_EvaluateCompletionConditions();

_CommandsCyclic();

IF FirstCycScan THEN
	_ComponentCyclic();
	FirstCycScan	:= FALSE;
END_IF

_UpdateBusyStatus();

_UpdateComponentStatus();

HMICommunication(); //Keeps the HMI data up to date, and processes requests from the HMI for this component
END_METHOD

END_FUNCTION_BLOCK

// Configuration/FB_CmdPermIntlkConfiguration
{attribute 'no_explicit_call' := 'do not call this POU directly'}
FUNCTION_BLOCK FB_CmdPermIntlkConfiguration EXTENDS FB_BaseStatic IMPLEMENTS I_CommandConfiguration, I_PermIntlkConfiguration
VAR
	PermIntlkConfiguration		: ST_PermIntlkConfiguration;
	CommandConfiguration		: ST_CommandConfiguration;
END_VAR

METHOD PROTECTED _InitializeReferences : BOOL
//Order is important!
BaseConfiguration.InstancePath 				REF= SUPER^.InstancePath;

PermIntlkConfiguration.BaseConfiguration 	REF= SUPER^.BaseConfiguration;
CommandConfiguration.BaseConfiguration		REF= SUPER^.BaseConfiguration;

CommandConfiguration.PermIntlkConfiguration REF= PermIntlkConfiguration;
                                	
_InitializeReferences 						:= TRUE; // apply at end of all reference initialization
END_METHOD

PROPERTY P_CommandConfiguration : REFERENCE TO ST_CommandConfiguration
GET
P_CommandConfiguration REF= CommandConfiguration;
END_GET
END_PROPERTY

PROPERTY P_PermIntlkConfiguration : REFERENCE TO ST_PermIntlkConfiguration
GET
P_PermIntlkConfiguration REF= PermIntlkConfiguration;
END_GET
END_PROPERTY

END_FUNCTION_BLOCK

// RingBuffer/POUs/FB_RingBufferICmd
{attribute 'no_explicit_call' := 'do not call this POU directly'}
FUNCTION_BLOCK FB_RingBufferICmd EXTENDS FB_RingBufferBase IMPLEMENTS I_RingBufferBase, I_RingBufferICmd
VAR
  Buffer              	: ARRAY[GPL_RingBuffer.MIN_NUMBER_OBJECTS..GPL_RingBuffer.MAX_NUMBER_OBJECTS] OF ST_SystimeICmd;
  LastObjRemoved		: ST_SystimeICmd;
  LastObjPeeked			: ST_SystimeICmd;
  LastObjRead			: ST_SystimeICmd;
END_VAR

METHOD ClearLastRemoved
MEMSET(destAddr := ADR(LastObjRemoved), fillByte := 16#00, n := RingBufferConfiguration.ByteCountOfDataObj);
END_METHOD

PROPERTY P_RingBufferStatus : REFERENCE TO ST_RingBufferStatus
GET
P_RingBufferStatus REF= SUPER^.RingBufferStatus;
END_GET
END_PROPERTY

METHOD PUBLIC RemoveObject
VAR_OUTPUT
    Error : BOOL;
END_VAR
VAR
    ByteSize : UDINT;
    Addr     : PVOID;
END_VAR
Error := FALSE;
ByteSize := RingBufferConfiguration.ByteCountOfDataObj;

IF RingBufferStatus.ObjectCountInBufferPrim = 0 THEN   (* nothing to pop *)
    Error := TRUE;
    RETURN;
END_IF;

Addr := pBufferStart +
        (RemoveIncrement MOD RingBufferStatus.BufferCapacity) * ByteSize;

IF Tc2_System.MEMMOVE(srcAddr := Addr, destAddr := ADR(LastObjRemoved), n := ByteSize) <> ByteSize THEN
    Error := TRUE;
    RETURN;
END_IF;
Tc2_System.MEMSET(destAddr := Addr, fillByte := 16#00, n := ByteSize);

(* advance remove side *)
RemoveIncrement := RemoveIncrement + 1;
RemoveIndex     := (RemoveIncrement MOD RingBufferStatus.BufferCapacity)
                 + GPL_RingBuffer.MIN_NUMBER_OBJECTS;
pRemove         := pBufferStart +
                   (RemoveIncrement MOD RingBufferStatus.BufferCapacity) * ByteSize;

(* counters / flags *)
RingBufferStatus.ObjectCountInBufferPrim := RingBufferStatus.ObjectCountInBufferPrim - 1;
IF RingBufferStatus.GlobalCounter > 0 THEN
    RingBufferStatus.GlobalCounter := RingBufferStatus.GlobalCounter - 1;
END_IF;

RingBufferStatus.ObjectWasRemovedPrimary := TRUE;

RingBufferStatus.Overwriting  := FALSE;                                 (* we freed space *)
RingBufferStatus.WillOverwrite :=                                     (* preview for next cycle *)
    (RingBufferStatus.ObjectCountInBufferPrim = RingBufferStatus.BufferCapacity);

(* derived *)
RingBufferStatus.BufferIsFullPrim :=
    (RingBufferStatus.ObjectCountInBufferPrim = RingBufferStatus.BufferCapacity);
RingBufferStatus.ByteCountInBufferPrim :=
    RingBufferStatus.ObjectCountInBufferPrim * ByteSize;
END_METHOD

METHOD PUBLIC AddObject
VAR_INPUT
    RefObject : REFERENCE TO ST_SystimeICmd;
END_VAR
VAR_OUTPUT
    Error : BOOL;
END_VAR
VAR
    ByteSize   : UDINT;
    ByteOffset : UDINT;
    WriteAddr  : PVOID;
END_VAR
Error := FALSE;
ByteSize := RingBufferConfiguration.ByteCountOfDataObj;

(* ---------- GUARDS ---------- *)
IF (RingBufferStatus.BufferCapacity = 0) OR (NOT __ISVALIDREF(RefObject)) THEN
    Error := TRUE;                           (* zero-capacity or bogus ref *)
    RETURN;
END_IF;

(* ---------- PREDICT / PREP ---------- *)
RingBufferStatus.WillOverwrite :=
    (RingBufferStatus.ObjectCountInBufferPrim >= RingBufferStatus.BufferCapacity);

ByteOffset := (WriteIncrement MOD RingBufferStatus.BufferCapacity) * ByteSize;
WriteAddr  := pBufferStart + ByteOffset;

(* ---------- WRITE ---------- *)
RefObject.systimestamp := Tc2_System.F_GetSystemTime();
IF Tc2_System.MEMMOVE(srcAddr := ADR(RefObject), destAddr := WriteAddr, n := ByteSize) <> ByteSize THEN
    Error := TRUE;
    RETURN;
END_IF;

(* ---------- ADVANCE WRITE POINTERS ---------- *)
WriteIncrement := WriteIncrement + 1;
WriteIndex := (WriteIncrement MOD RingBufferStatus.BufferCapacity)
            + GPL_RingBuffer.MIN_NUMBER_OBJECTS;

(* ---------- COUNTERS & FLAGS ---------- *)
IF RingBufferStatus.WillOverwrite THEN
    (* buffer is full – push remove side forward one slot *)
    RemoveIncrement := RemoveIncrement + 1;
    pRemove := pBufferStart
             + (RemoveIncrement MOD RingBufferStatus.BufferCapacity) * ByteSize;
    RingBufferStatus.Overwriting := TRUE;              (* occurred *this* cycle *)
ELSE
    RingBufferStatus.ObjectCountInBufferPrim := RingBufferStatus.ObjectCountInBufferPrim + 1;
    RingBufferStatus.GlobalCounter           := RingBufferStatus.GlobalCounter + 1;
    RingBufferStatus.Overwriting             := FALSE;
END_IF;

RingBufferStatus.ObjectWasAddedPrimary := TRUE;

(* ---------- STATE FOR NEXT SCAN ---------- *)
RingBufferStatus.WillOverwrite :=
    (RingBufferStatus.ObjectCountInBufferPrim >= RingBufferStatus.BufferCapacity);

(* ---------- DERIVED VALUES ---------- *)
RingBufferStatus.BufferIsFullPrim :=
    (RingBufferStatus.ObjectCountInBufferPrim = RingBufferStatus.BufferCapacity);
RingBufferStatus.ByteCountInBufferPrim :=
    RingBufferStatus.ObjectCountInBufferPrim * ByteSize;
END_METHOD

PROPERTY P_Buffer : REFERENCE TO ARRAY[GPL_RingBuffer.MIN_NUMBER_OBJECTS..GPL_RingBuffer.MAX_NUMBER_OBJECTS] OF ST_SystimeICmd;
GET
P_Buffer REF= Buffer;
END_GET
END_PROPERTY

PROPERTY P_LastObjectPeeked : REFERENCE TO ST_SystimeICmd
GET
P_LastObjectPeeked REF= LastObjPeeked;
END_GET
END_PROPERTY

PROPERTY P_LastObjectRead : REFERENCE TO ST_SystimeICmd
GET
P_LastObjectRead REF= LastObjRead;
END_GET
END_PROPERTY

PROPERTY P_LastObjectRemoved : REFERENCE TO ST_SystimeICmd
GET
P_LastObjectRemoved REF= LastObjRemoved;
END_GET
END_PROPERTY

METHOD PUBLIC PeekObject : ST_SystimeICmd
PeekIndex := (RemoveIncrement MOD SUPER^.RingBufferStatus.BufferCapacity) + GPL_RingBuffer.MIN_NUMBER_OBJECTS;
PeekAddr := pBufferStart + (PeekIndex - GPL_RingBuffer.MIN_NUMBER_OBJECTS) * RingBufferConfiguration.ByteCountOfDataObj;

// Step 2: Conditional peek (non-mutating)
IF SUPER^.RingBufferStatus.GlobalCounter > 0 THEN
    SUPER^.RingBufferStatus.CountBytesPeeked := Tc2_System.MEMMOVE(
        srcAddr := PeekAddr,
        destAddr := ADR(LastObjPeeked),
        n := RingBufferConfiguration.ByteCountOfDataObj
    );

    IF SUPER^.RingBufferStatus.CountBytesPeeked > 0 THEN
        RingBufferStatus.ObjectWasPeekedPrimary := TRUE;
		PeekObject	:= LastObjPeeked;
    END_IF
ELSE
    RingBufferStatus.ObjectWasPeekedPrimary := FALSE;
    //LastObjPeeked.stringval := '';
END_IF
END_METHOD

METHOD ReadObject : ST_SystimeICmd
VAR_OUTPUT
  Error : BOOL;
END_VAR
// Step 1: Check if buffer has data
IF SUPER^.RingBufferStatus.GlobalCounter > 0 THEN

    // Step 2: Calculate read offset and pointer
    RingBufferConfiguration.ReadByteOffset := (RemoveIncrement MOD RingBufferStatus.BufferCapacity) * RingBufferConfiguration.ByteCountOfDataObj;
    ReadAddr := pBufferStart + RingBufferConfiguration.ReadByteOffset;

    // Step 3: Read memory
    SUPER^.RingBufferStatus.CountBytesRead := Tc2_System.MEMMOVE(
        srcAddr := ReadAddr,
        destAddr := ADR(LastObjRead),
        n := RingBufferConfiguration.ByteCountOfDataObj
    );

    // Step 4: Handle result
    IF SUPER^.RingBufferStatus.CountBytesRead = RingBufferConfiguration.ByteCountOfDataObj THEN
        RingBufferStatus.ObjectWasReadPrimary := TRUE;

        RemoveIncrement := RemoveIncrement + 1;

        // Update index and pRemove based on RemoveIncrement
        RemoveIndex := (RemoveIncrement MOD RingBufferStatus.BufferCapacity)
                       + GPL_RingBuffer.MIN_NUMBER_OBJECTS;

        pRemove := pBufferStart + 
                   (RemoveIncrement MOD RingBufferStatus.BufferCapacity) * RingBufferConfiguration.ByteCountOfDataObj;

        SUPER^.RingBufferStatus.GlobalCounter := SUPER^.RingBufferStatus.GlobalCounter - 1;
    ELSE
        RingBufferStatus.ObjectWasReadPrimary := FALSE;
        //LastObjRead.stringval := ''; // 🛠 Corrected
        Error := TRUE;
    END_IF
ELSE
    RingBufferStatus.ObjectWasReadPrimary := FALSE;
    //LastObjRead.stringval := ''; // 🛠 Corrected
    Error := TRUE;
END_IF

UpdateObjectCtInBuffers();
END_METHOD

METHOD PROTECTED UpdateRemovePointer
VAR_INPUT
  pRemovePtr  : PVOID;
END_VAR
pRemove := ADR(Buffer[RemoveIndex]);

pRemoveUpdated  := TRUE;
END_METHOD

METHOD PROTECTED UpdateWritePointer
VAR_INPUT
  pWritePtr  : PVOID;
END_VAR
IF (WriteIndex = GPL_RingBuffer.MIN_NUMBER_OBJECTS) THEN
  pWrite        := ADR(Buffer[GPL_RingBuffer.MIN_NUMBER_OBJECTS]);
ELSIF (WriteIndex > GPL_RingBuffer.MIN_NUMBER_OBJECTS) AND 
  (WriteIndex <= GPL_RingBuffer.MAX_NUMBER_OBJECTS) THEN
  pWrite        := IncrementPointer(pPointer  := pWrite, ByteCtIncrement := RingBufferConfiguration.ByteCountOfDataObj);
END_IF

pWriteUpdated   := TRUE;
END_METHOD

(* Basic component initialization logic*)
METHOD PROTECTED _Initialize : BOOL
VAR
	InterimInit : BOOL;
END_VAR
InterimInit := _InitializeChildrenDependencies();

InterimInit	:= _InitializeReferences();

IF NOT InterimInit THEN
	IF SUPER^.BaseConfiguration.LogTraceConfiguration.What.xLogToEventLogger THEN
		TraceWithSeverity(Message := Tc2_Standard.CONCAT('Initialization Failed at ', __POUNAME()), Severity := Global.TcEventSeverity.Error);
	END_IF
END_IF

RingBufferStatus.BufferCapacity  := (GPL_RingBuffer.MAX_NUMBER_OBJECTS - GPL_RingBuffer.MIN_NUMBER_OBJECTS) +1;

RemoveIndex  := GPL_RingBuffer.MIN_NUMBER_OBJECTS;
PeekIndex	 := GPL_RingBuffer.MIN_NUMBER_OBJECTS;

pBufferStart	:= ADR(Buffer[GPL_RingBuffer.MIN_NUMBER_OBJECTS]);

RingBufferConfiguration.ByteCountOfDataObj      := SIZEOF(Buffer[GPL_RingBuffer.MIN_NUMBER_OBJECTS]);

IF (pWrite = Tc3_Module.NULL) THEN
  pWrite  := ADR(Buffer[GPL_RingBuffer.MIN_NUMBER_OBJECTS]);
END_IF

IF (pRemove = Tc3_Module.NULL) THEN
  pRemove  := ADR(Buffer[GPL_RingBuffer.MIN_NUMBER_OBJECTS]);
END_IF

InterimInit	:= _SetDependencyConfiguration();

_Initialize 	:= InterimInit;
END_METHOD

METHOD ClearBuffer
MEMSET(destAddr := ADR(Buffer[GPL_RingBuffer.MIN_NUMBER_OBJECTS]), fillByte := 16#00, n := (RingBufferConfiguration.ByteCountOfDataObj*SUPER^.RingBufferStatus.BufferCapacity));

WriteIncrement := 0;
RemoveIncrement := 0;
SUPER^.RingBufferStatus.GlobalCounter := 0;
pWrite := ADR(Buffer[GPL_RingBuffer.MIN_NUMBER_OBJECTS]);
pRemove := ADR(Buffer[GPL_RingBuffer.MIN_NUMBER_OBJECTS]);
UpdateObjectCtInBuffers();
END_METHOD

END_FUNCTION_BLOCK

// RingBuffer/POUs/FB_RingBufferBase
FUNCTION_BLOCK ABSTRACT FB_RingBufferBase EXTENDS FB_BaseStatic
VAR
	RingBufferConfiguration    		: ST_RingBufferCfg;
	pRemove        					: PVOID;
	pWrite         					: PVOID;
	pBufferStart					: PVOID;
	RemoveAddr 						: PVOID;
	PeekAddr						: PVOID;
	ReadAddr						: PVOID;
	pRemoveUpdated 					: BOOL;
	pWriteUpdated  					: BOOL;
	WriteIncrement 					: UDINT;
	RemoveIncrement					: UDINT;
	WriteIndex     					: UDINT;
	RemoveIndex    					: UDINT;
	PeekIndex						: UDINT;
	ReadIndex						: UDINT;
	RingBufferStatus				: ST_RingBufferStatus;
END_VAR

(* Basic component initialization logic*)
METHOD PROTECTED _Initialize : BOOL
VAR
	InterimInit : BOOL;
END_VAR
// Initialize children dependencies first
InterimInit := _InitializeChildrenDependencies();
IF NOT InterimInit THEN
	IF BaseConfiguration.LogTraceConfiguration.What.xLogToEventLogger AND NOT BaseStatus.LogTraceStatus.InitChildrenFailureShown THEN
		TraceWithSeverity(Message := Tc2_Standard.CONCAT('_InitializeChildrenDependencies Failed at ', __POUNAME()), Severity := Global.TcEventSeverity.Error);
		BaseStatus.LogTraceStatus.InitChildrenFailureShown := TRUE;
	END_IF
	_Initialize := FALSE;
	RETURN;
END_IF

// Initialize references second
InterimInit := _InitializeReferences();
IF NOT InterimInit THEN
	IF BaseConfiguration.LogTraceConfiguration.What.xLogToEventLogger AND NOT BaseStatus.LogTraceStatus.InitReferencesFailureShown THEN
		TraceWithSeverity(Message := Tc2_Standard.CONCAT('_InitializeReferences Failed at ', __POUNAME()), Severity := Global.TcEventSeverity.Error);
		BaseStatus.LogTraceStatus.InitReferencesFailureShown := TRUE;
	END_IF
	_Initialize := FALSE;
	RETURN;
END_IF

// Set buffer-specific initialization values
RingBufferStatus.BufferCapacity := (GPL_RingBuffer.MAX_NUMBER_OBJECTS - GPL_RingBuffer.MIN_NUMBER_OBJECTS) + 1;
RemoveIndex := GPL_RingBuffer.MIN_NUMBER_OBJECTS;
PeekIndex := GPL_RingBuffer.MIN_NUMBER_OBJECTS;

// Set dependency configuration last
InterimInit := _SetDependencyConfiguration();
IF NOT InterimInit THEN
	IF BaseConfiguration.LogTraceConfiguration.What.xLogToEventLogger AND NOT BaseStatus.LogTraceStatus.InitDependencyConfigFailureShown THEN
		TraceWithSeverity(Message := Tc2_Standard.CONCAT('_SetDependencyConfiguration Failed at ', __POUNAME()), Severity := Global.TcEventSeverity.Error);
		BaseStatus.LogTraceStatus.InitDependencyConfigFailureShown := TRUE;
	END_IF
	_Initialize := FALSE;
	RETURN;
END_IF

// All initialization steps succeeded
_Initialize := TRUE;
END_METHOD

METHOD PROTECTED _InitializeReferences : BOOL
//Order is important!
BaseConfiguration.InstancePath 				REF= SUPER^.InstancePath;

RingBufferConfiguration.BaseConfiguration	REF= SUPER^.BaseConfiguration;

RingBufferStatus.BaseStatus					REF= SUPER^.BaseStatus;

_InitializeReferences 						:= TRUE;
END_METHOD

METHOD PROTECTED UpdateObjectCtInBuffers
RingBufferStatus.BufferIsFullPrim :=
    (RingBufferStatus.ObjectCountInBufferPrim = RingBufferStatus.BufferCapacity);
RingBufferStatus.ByteCountInBufferPrim :=
    RingBufferStatus.ObjectCountInBufferPrim * RingBufferConfiguration.ByteCountOfDataObj;
END_METHOD

PROPERTY P_ObjCountInBuffer : ULINT
GET
P_ObjCountInBuffer  := RingBufferStatus.ObjectCountInBufferPrim;
END_GET
END_PROPERTY

PROPERTY P_ObjectWasAdded : REFERENCE TO BOOL
GET
//P_ObjectWasAdded REF= RingBufferStatus.ObjectWasAddedPrimary;
P_ObjectWasAdded REF= RingBufferStatus.ObjectWasAddedPrimary;
END_GET
END_PROPERTY

PROPERTY P_ObjectWasPeeked : REFERENCE TO BOOL
GET
P_ObjectWasPeeked REF= RingBufferStatus.ObjectWasPeekedPrimary;
END_GET
END_PROPERTY

PROPERTY P_ObjectWasRead : REFERENCE TO BOOL
GET
P_ObjectWasRead REF= RingBufferStatus.ObjectWasReadPrimary;
END_GET
END_PROPERTY

PROPERTY P_ObjectWasRemoved : REFERENCE TO BOOL
GET
P_ObjectWasRemoved REF= RingBufferStatus.ObjectWasRemovedPrimary;
END_GET
END_PROPERTY

METHOD ABSTRACT ClearLastRemoved
END_METHOD

METHOD PROTECTED IncrementPointer : ULINT
VAR_INPUT
  pPointer        : PVOID;
  ByteCtIncrement : ULINT; 
END_VAR
IncrementPointer :=
    WrapPointer(
        BasePtr    := pBufferStart,
        CurrentPtr := pPointer + ByteCtIncrement,
        ByteSize   := RingBufferConfiguration.ByteCountOfDataObj,
        Capacity   := RingBufferStatus.BufferCapacity );
END_METHOD

METHOD PROTECTED ABSTRACT UpdateRemovePointer
VAR_INPUT
  pRemovePtr  : PVOID;
END_VAR
END_METHOD

METHOD PROTECTED ABSTRACT UpdateWritePointer
VAR_INPUT
  pWritePtr  : PVOID;
END_VAR
END_METHOD

METHOD ClearStatusFlagAdded
RingBufferStatus.ObjectWasAddedPrimary := FALSE;
END_METHOD

METHOD ClearStatusFlagPeeked
RingBufferStatus.ObjectWasPeekedPrimary := FALSE;
END_METHOD

METHOD ClearStatusFlagRead
RingBufferStatus.ObjectWasReadPrimary := FALSE;
END_METHOD

METHOD ClearStatusFlagRemoved
RingBufferStatus.ObjectWasRemovedPrimary := FALSE;
END_METHOD

METHOD ClearStatusFlags
ClearStatusFlagAdded();
ClearStatusFlagPeeked();
ClearStatusFlagRead();
ClearStatusFlagRemoved();
END_METHOD

METHOD PRIVATE WrapPointer : PVOID
VAR_INPUT
    BasePtr        : PVOID;   (* pBufferStart *)
    CurrentPtr     : PVOID;   (* pWrite or pRemove *)
    ByteSize       : UDINT;   (* ByteCountOfDataObj *)
    Capacity       : UDINT;   (* BufferCapacity *)
END_VAR
VAR
    Offset : ULINT;
END_VAR
Offset := (CurrentPtr - BasePtr) MOD (ByteSize * Capacity);
WrapPointer := BasePtr + Offset;
END_METHOD

END_FUNCTION_BLOCK

// Hashing/POUs/FB_Hash_djb2
{attribute 'no_explicit_call' := 'do not call this POU directly'}
FUNCTION_BLOCK FB_Hash_djb2 EXTENDS FB_BaseStatic IMPLEMENTS I_HashFunction
VAR CONSTANT
	djb2Init				: UDINT := 5381;
END_VAR
VAR
	h 						: UDINT := djb2Init;
	i 						: INT;
	b 						: BYTE;
	_HashTable				: I_HashTableBase;
END_VAR

METHOD Hash : UINT
VAR_INPUT
    Key 		: T_MaxString;
	Capacity 	: UINT := GPL_HashTable.INDEX_MAX;
END_VAR
// Check basic capacity validity
IF (Capacity = 0) THEN
    Hash := UINT#65535;
    IF BaseConfiguration.LogTraceConfiguration.What.xLogToEventLogger THEN
        TraceWithSeverity('Hash(): Capacity must be non-zero', Severity := Global.TcEventSeverity.Error);
    END_IF
    RETURN;
END_IF

// Skip HashTable validation - let it work standalone
// Power-of-2 validation can be handled by the caller if needed

h := djb2Init;
//--- djb2 core: h = ((h << 5) + h) + b
FOR i := 1 TO LEN(Key) DO
    b := TO_BYTE(Key[i]);
    h := Tc2_System.SHL32(h, 5) + h + BYTE_TO_UDINT(b);
END_FOR

//--- Fold hash into table range [0 .. Capacity-1]
// Use modulo for non-power-of-2 capacities, but prefer masking for power-of-2
IF F_IsPowerOfTwo_UINT(Value := Capacity) THEN
    Hash := UDINT_TO_UINT(h AND UINT_TO_UDINT(Capacity - 1));
ELSE
    Hash := UDINT_TO_UINT(h MOD UINT_TO_UDINT(Capacity));
END_IF
END_METHOD

PROPERTY P_TP_HashTableStatus : REFERENCE TO ST_HashTableStatus
GET
// Return invalid reference to prevent page faults
// The caller should check __ISVALIDREF before using this property
END_GET
END_PROPERTY

END_FUNCTION_BLOCK

// Hashing/ITFs/I_HashFunction
INTERFACE I_HashFunction EXTENDS I_BaseStatic

METHOD Hash : UINT
VAR_INPUT
	Key : T_MaxString;
	Capacity : UINT;
END_VAR
END_METHOD

END_INTERFACE

// Hashing/ITFs/I_HashTableBase
INTERFACE I_HashTableBase EXTENDS I_BaseStatic

//— Completely clear all entries
METHOD Clear
END_METHOD

//— Lookup name → index
METHOD PUBLIC GetIndex : UINT
VAR_INPUT
  NameIn : T_MaxString;
END_VAR
END_METHOD

//— Insert or overwrite an entry; auto‐rehash if load too high
METHOD PUBLIC Insert
VAR_INPUT
	NameIn : T_MaxString;
	IdxIn  : UINT;
END_VAR
END_METHOD

PROPERTY P_HashTableStatus : REFERENCE TO ST_HashTableStatus
GET
END_GET
END_PROPERTY

END_INTERFACE

// Functions/Numbers/F_IsPowerOfTwo_UINT
FUNCTION F_IsPowerOfTwo_UINT : BOOL
VAR_INPUT
    Value : UINT;    // Supports signed values
END_VAR
VAR
    i        : UINT;
    shifted  : DWORD;
END_VAR

// Negative numbers and 0 are not powers of two
IF Value <= 0 THEN
    F_IsPowerOfTwo_uINT := FALSE;
    RETURN;
END_IF

// Try all bit positions 0..30 (since SHL32 on 1<<31 gives negative result)
FOR i := 0 TO 30 DO
    shifted := Tc2_System.SHL32(1, UINT_TO_SINT(i));
    IF Value = shifted THEN
        F_IsPowerOfTwo_uINT := TRUE;
        RETURN;
    END_IF
END_FOR

// No match → not a power of two
F_IsPowerOfTwo_UINT := FALSE;

END_FUNCTION

// Hashing/POUs/FB_HashTable
(*-------------------------------------------------------------------------                                          	
(   Builds and maintains a hash‐map from POU name (string) → index (UINT) 
(-------------------------------------------------------------------------*)
{attribute 'no_explicit_call' := 'do not call this POU directly'}
FUNCTION_BLOCK FB_HashTable EXTENDS FB_BaseStatic IMPLEMENTS I_HashTableBase, I_HashTableConfiguration

VAR
	HashTableConfiguration	: ST_HashTableConfiguration;	
	HashTableStatus			: ST_HashTableStatus;
	Keys        			: ARRAY[GPL_HashTable.INDEX_MIN..GPL_HashTable.INDEX_MAX] OF T_MaxString;
	Values       			: ARRAY[GPL_HashTable.INDEX_MIN..GPL_HashTable.INDEX_MAX] OF UINT;
	_HashFunction			: I_HashFunction;
END_VAR

VAR CONSTANT
	EMPTY_KEY				: T_MaxString := '';        // unused slot sentinel
	TOMBSTONE				: T_MaxString := '<DEL>';   // delete‐marker sentinel
END_VAR

VAR
	h           			: UDINT;  // raw 32-bit hash code from the hash function.
	idx         			: UINT; //the current bucket index you’re probing into (i.e. “where in the array we are right now”).
	probeCount  			: UINT; //a loop counter to make sure you don’t probe more times than the table’s size (and thus get stuck in an infinite loop).
	keyAtIdx    			: T_MaxString; //keyAtIdx: a local copy of Keys[idx] so you can compare against the lookup name or check for an empty slot without repeatedly indexing into the array.
END_VAR

//— Completely clear all entries
METHOD Clear
_InitializeHashTable();
END_METHOD

METHOD PUBLIC GetIndex : UINT
VAR_INPUT
    NameIn : T_MaxString;
END_VAR
GetIndex := UINT#65535;

IF _HashFunction = 0 THEN
    IF HashTableConfiguration.BaseConfiguration.LogTraceConfiguration.What.xLogToEventLogger THEN
        TraceWithSeverity(Message := 'Hash Function Interface not provided - Returning!', Severity := Global.TcEventSeverity.Error);
    END_IF
    RETURN; // Prevent invalid use
END_IF

h := _HashFunction.Hash(Key := NameIn, Capacity := HashTableConfiguration.Capacity);
// The Hash function already returns a value in range [0..Capacity-1], so use it directly
idx := UDINT_TO_UINT(h);


FOR probeCount := 0 TO HashTableConfiguration.Capacity - 1 DO
    keyAtIdx := Keys[idx];

    IF keyAtIdx = NameIn THEN
        GetIndex := Values[idx];
        RETURN;
    ELSIF keyAtIdx = EMPTY_KEY THEN
        RETURN;
    END_IF

    idx := (idx + 1) MOD HashTableConfiguration.Capacity;
END_FOR
END_METHOD

//— Insert or overwrite an entry; auto‐rehash if load too high
METHOD PUBLIC Insert
VAR_INPUT
	NameIn : T_MaxString;
	IdxIn  : UINT;
END_VAR
// Defensive check
IF _HashFunction = 0 THEN
	IF HashTableConfiguration.BaseConfiguration.LogTraceConfiguration.What.xLogToEventLogger THEN
		TraceWithSeverity(Message := 'Hash Function Interface not provided - Returning!', Severity := Global.TcEventSeverity.Error);
	END_IF
	RETURN;
END_IF

// Compute hash
h := _HashFunction.Hash(Key := NameIn, Capacity := HashTableConfiguration.Capacity);

// The Hash function already returns a value in range [0..Capacity-1], so use it directly
idx := UDINT_TO_UINT(h);

// Linear probing to find insert position
FOR probeCount := 0 TO HashTableConfiguration.Capacity - 1 DO
	keyAtIdx := Keys[idx];

	IF keyAtIdx = NameIn THEN
		// Overwrite existing key
		Values[idx] := IdxIn;
		RETURN;
	ELSIF keyAtIdx = EMPTY_KEY THEN
		// Insert new entry
		Keys[idx] := NameIn;
		Values[idx] := IdxIn;
		HashTableStatus.Count := HashTableStatus.Count + 1;
		EXIT;
	END_IF

	// Next probe
	idx := (idx + 1) MOD HashTableConfiguration.Capacity;
END_FOR

// Optional: log full-table condition
// Trace('Hash table insert failed: table full.');

// Check load factor to optionally trigger rehash

IF HashTableStatus.Capacity <> 0 THEN
	HashTableStatus.LoadFactor := (UINT_TO_REAL(HashTableStatus.Count) / UINT_TO_REAL(HashTableStatus.Capacity));
END_IF

IF __ISVALIDREF(HashTableStatus.LoadFactor) THEN
	IF HashTableStatus.LoadFactor > HashTableConfiguration.LoadFactor THEN
		IF HashTableConfiguration.BaseConfiguration.LogTraceConfiguration.What.xLogToEventLogger THEN
			TraceWithSeverity(Message := 'Hash Table Load Factor exceeded; recommend Rehash!', Severity := Global.TcEventSeverity.Warning);
		END_IF
		// _Rehash();
	END_IF
END_IF
END_METHOD

PROPERTY P_HashTableStatus : REFERENCE TO ST_HashTableStatus
GET
P_HashTableStatus REF= HashTableStatus;
END_GET
END_PROPERTY

PROPERTY P_HashTableConfiguration : REFERENCE TO ST_HashTableConfiguration
GET
P_HashTableConfiguration REF= HashTableConfiguration;
END_GET
END_PROPERTY

METHOD PROTECTED _Initialize : BOOL
VAR
	InterimInit : BOOL;
END_VAR
SUPER^._Initialize();

InterimInit	:= _InitializeHashTable();

//Check if capacity is a power of 2
IF NOT F_IsPowerOfTwo_UINT(Value := HashTableConfiguration.Capacity) THEN
	IF HashTableConfiguration.BaseConfiguration.LogTraceConfiguration.What.xLogToEventLogger THEN
		TraceWithSeverity(Message := 'Make Hash Table array size a power of 2!', Severity := Global.TcEventSeverity.Error);
	END_IF
ELSE
	HashTableStatus.HashTableIsPowerOf2 := TRUE;
END_IF

InterimInit	:= _SetDependencyConfiguration();

_Initialize := TRUE;
END_METHOD

METHOD PROTECTED _InitializeChildrenDependencies : BOOL
IF _HashFunction <> 0 THEN
	_HashFunction.Initialize();
END_IF

_InitializeChildrenDependencies := TRUE;
END_METHOD

METHOD PROTECTED _InitializeHashTable : BOOL
VAR
  i : DINT;
  actualCapacity : UINT;
END_VAR
//— Initialize (or re‐init) the table
// Calculate actual capacity from array bounds
actualCapacity := DINT_TO_UINT(UPPER_BOUND(Keys,1) - LOWER_BOUND(Keys,1) + 1);
HashTableConfiguration.Capacity := actualCapacity;

//FOR i := LOWER_BOUND(Keys,1) TO UPPER_BOUND(Keys,1) DO
MEMSET(fillByte := STRING_TO_BYTE(EMPTY_KEY), destAddr := ADR(Keys[GPL_HashTable.INDEX_MIN]), n := (actualCapacity*SIZEOF(Keys[GPL_HashTable.INDEX_MIN])));
MEMSET(fillByte := 16#00, destAddr := ADR(Values[GPL_HashTable.INDEX_MIN]), n := actualCapacity*SIZEOF(Values[GPL_HashTable.INDEX_MIN]));
//END_FOR
HashTableStatus.Count 		:= 0;

_InitializeHashTable	:= TRUE;
END_METHOD

METHOD PROTECTED _InitializeReferences : BOOL
//Order is important!
BaseConfiguration.InstancePath 				REF= InstancePath;

HashTableConfiguration.BaseConfiguration	REF= SUPER^.BaseConfiguration;

HashTableStatus.BaseStatus					REF= SUPER^.BaseStatus;

HashTableStatus.Capacity					REF= HashTableConfiguration.Capacity;

HashTableStatus.LoadFactor					REF= HashTableConfiguration.LoadFactor;

_InitializeReferences 						:= TRUE; // apply at end of all reference initialization
END_METHOD

METHOD InjectHashFunction : BOOL
VAR_INPUT
	iHashFunction			: I_HashFunction;
END_VAR
THIS^._HashFunction := iHashFunction;
END_METHOD

END_FUNCTION_BLOCK

// Hashing/ITFs/I_HashTableConfiguration
INTERFACE I_HashTableConfiguration EXTENDS I_BaseStatic

PROPERTY P_HashTableConfiguration : REFERENCE TO ST_HashTableConfiguration
GET
END_GET
END_PROPERTY

END_INTERFACE

// ControlMode/POUs/FB_ControlMode
{attribute 'no_explicit_call' := 'do not call this POU directly'}
FUNCTION_BLOCK FB_ControlMode EXTENDS FB_Component<GC_ControlMode.INDEX_COMMAND_MIN,GC_ControlMode.INDEX_COMMAND_MAX> IMPLEMENTS I_ControlMode
VAR
	ControlMode	: DINT;
END_VAR

METHOD ChangeMode : I_ControlMode
VAR_INPUT
	DesiredMode	: DINT;
END_VAR
VAR
	CommandIndex				: DINT; // FOR Loop, etc.
END_VAR
//TODO
//Check Permissive
FOR CommandIndex := LOWER_BOUND(SUPER^.CommandPermIntlkConfiguration,1) TO UPPER_BOUND(SUPER^.CommandPermIntlkConfiguration,1) BY 1 DO

	IF SUPER^.CommandPermIntlkConfiguration[CommandIndex].P_CommandConfiguration.CommandDescription = F_GetLastWordInString(__POUNAME()) THEN
		ExecuteCommand(CmdIndex := SUPER^.CommandPermIntlkConfiguration[CommandIndex].P_CommandConfiguration.CommandIndex);
	END_IF

	IF SUPER^.iCommands[CommandIndex].P_CommandStatus.Result = E_CommandResult.Ok THEN
		ControlMode	:= DesiredMode;
	END_IF
	
END_FOR

ChangeMode	:= THIS^;
END_METHOD

{warning 'Add property implementation'}
PROPERTY P_ControlMode : DINT
GET
P_ControlMode := ControlMode;
END_GET
END_PROPERTY

METHOD PROTECTED _EvaluateCompletionConditions : BOOL
END_METHOD

(* Example implementation from FB_Actuator:
IF ActuatorStatus.ExtendOutput AND NOT ActuatorStatus.RetractOutput THEN
	ActuatorStatus.ActuatorState	:= E_ActuatorState.Extended;
ELSIF ActuatorStatus.RetractOutput AND NOT ActuatorStatus.ExtendOutput THEN
	ActuatorStatus.ActuatorState	:= E_ActuatorState.Retracted;
ELSE
	ActuatorStatus.ActuatorState	:= E_ActuatorState.Indeterminate;
END_IF

_UpdateComponentStatus := THIS^;*)
METHOD PROTECTED _UpdateComponentStatus : I_ComponentFull
END_METHOD

METHOD InjectControlModeCmdPermIntlkConfigurations
VAR_INPUT
	SystemPermIntlk				: I_PermIntlk;
	ControlMode					: I_ControlMode;
	CommandConfiguration		: ARRAY[GC_ControlMode.INDEX_COMMAND_MIN..GC_ControlMode.INDEX_COMMAND_MAX] OF I_CommandConfiguration;
	PermIntlkConfiguration		: ARRAY[GC_ControlMode.INDEX_COMMAND_MIN..GC_ControlMode.INDEX_COMMAND_MAX] OF I_PermIntlkConfiguration;
END_VAR
InjectSystemInterfaces(ControlMode := ControlMode, SystemPermIntlk := SystemPermIntlk);

// Copy config data into CommandPermIntlkConfiguration
FOR SUPER^.CommandIndexCyclic := LOWER_BOUND(CommandConfiguration,1) TO MIN(UPPER_BOUND(CommandConfiguration,1),UPPER_BOUND(SUPER^.CommandPermIntlkConfiguration,1)) BY 1 DO
	SUPER^.CommandPermIntlkConfiguration[SUPER^.CommandIndexCyclic].P_CommandConfiguration :=
		CommandConfiguration[SUPER^.CommandIndexCyclic].P_CommandConfiguration;
	SUPER^.CommandPermIntlkConfiguration[SUPER^.CommandIndexCyclic].P_PermIntlkConfiguration :=
		PermIntlkConfiguration[SUPER^.CommandIndexCyclic].P_PermIntlkConfiguration;
	SUPER^.iCommands[SUPER^.CommandIndexCyclic] := SUPER^.Commands[SUPER^.CommandIndexCyclic]; // Initialize interface to command implementation
END_FOR
END_METHOD

END_FUNCTION_BLOCK

// Functions/Strings/F_GetLastWordInString
FUNCTION F_GetLastWordInString : Tc2_System.T_MaxString
VAR_INPUT
    sInput : Tc2_System.T_MaxString; // Input string
    ReturnChar       : BYTE := 46; // ASCII value of "."
END_VAR
VAR
    i           : INT;
    strLength   : INT;
    resultStr   : Tc2_System.T_MaxString;
    arrInput    : ARRAY[0..255] OF BYTE;
END_VAR

strLength := LEN(sInput);
arrInput := Tc2_Utilities.MAXSTRING_TO_BYTEARR(sInput); // Convert to BYTE array

// If last char is '.', return empty string
IF arrInput[strLength] = ReturnChar THEN
	F_GetLastWordInString := '';
	RETURN;
END_IF

// Build result by prepending characters from right to left
resultStr := '';
FOR i := strLength TO 1 BY -1 DO
	IF arrInput[i] = ReturnChar THEN
		EXIT;
	END_IF
	resultStr := Tc2_Standard.CONCAT(Tc2_System.F_ToCHR(arrInput[i]), resultStr);
END_FOR

F_GetLastWordInString := resultStr;

END_FUNCTION

// Debounce/FB_Debounce
{attribute 'no_explicit_call' := 'do not call this POU directly'}
FUNCTION_BLOCK FB_Debounce EXTENDS FB_BaseCyclic IMPLEMENTS I_DebounceConfiguration, I_Debounce
VAR
	DebounceConfiguration	: ST_DebounceConfiguration;
	DebounceStatus			: ST_DebounceStatus;

	TimerOn 				: Tc2_Standard.TON;
	TimerOff 				: Tc2_Standard.TOF;
END_VAR

METHOD PROTECTED _InitializeReferences : BOOL
//Order is important!
BaseConfiguration.InstancePath 	REF= InstancePath;

IF BaseConfiguration.LogTraceConfiguration.When = E_LogTraceWhen.xRunOnInitOnly AND_THEN
   BaseConfiguration.LogTraceConfiguration.What.xLogToEventLogger THEN
	TraceWithSeverity(Message := Tc2_Standard.CONCAT('If you created new data structures, they may not have valid pointer references; Check ', __POUNAME()), Severity := Global.TcEventSeverity.Warning);
END_IF

DebounceConfiguration.BaseConfiguration		REF= SUPER^.BaseConfiguration;

DebounceStatus.BaseStatus					REF= SUPER^.BaseStatus;

IF DebounceConfiguration.BaseConfiguration.InSimulation THEN
	DebounceStatus.RefRawSignal				REF= DebounceConfiguration.xSimSignal;
ELSE
	DebounceStatus.RefRawSignal				REF= DebounceConfiguration.xRawSignal;
END_IF

_InitializeReferences 						:= TRUE; // apply at end of all reference initialization
END_METHOD

METHOD CyclicLogic
SUPER^.CyclicLogic();

// Standard debounce: chain TON (rising edge delay) → TOF (falling edge delay)
// When InSimulation=TRUE, use P_RawSignal property to set xRawSignal programmatically
// When InSimulation=FALSE, xRawSignal reads from hardware I/O (AT %I*)

TimerOn(IN := P_RawSignal, PT := DebounceConfiguration.tOnDelay);
TimerOff(IN := TimerOn.Q, PT := DebounceConfiguration.tOffDelay);

DebounceStatus.DebouncedSignal := TimerOff.Q;

// Edge detection on debounced output
DebounceStatus.rtOutput(CLK := DebounceStatus.DebouncedSignal);
DebounceStatus.ftOutput(CLK := DebounceStatus.DebouncedSignal);

DebounceStatus.QRise := DebounceStatus.rtOutput.Q;
DebounceStatus.QFall := DebounceStatus.ftOutput.Q;
END_METHOD

PROPERTY P_DebounceConfiguration : REFERENCE TO ST_DebounceConfiguration
GET
P_DebounceConfiguration REF= DebounceConfiguration;
END_GET
END_PROPERTY

PROPERTY P_DebounceStatus : REFERENCE TO ST_DebounceStatus
GET
P_DebounceStatus REF= DebounceStatus;
END_GET
END_PROPERTY

PROPERTY P_RawSignal : BOOL
GET
IF DebounceConfiguration.BaseConfiguration.InSimulation THEN
	P_RawSignal := DebounceConfiguration.xSimSignal;
ELSE
	P_RawSignal := DebounceConfiguration.xRawSignal;
END_IF
END_GET
SET
IF DebounceConfiguration.BaseConfiguration.InSimulation THEN
	DebounceConfiguration.xSimSignal := P_RawSignal;
ELSE
	DebounceConfiguration.xRawSignal := P_RawSignal;
END_IF
END_SET
END_PROPERTY

END_FUNCTION_BLOCK

// Debounce/I_DebounceConfiguration
INTERFACE I_DebounceConfiguration EXTENDS __SYSTEM.IQueryInterface

PROPERTY P_DebounceConfiguration : REFERENCE TO ST_DebounceConfiguration
GET
END_GET
END_PROPERTY

END_INTERFACE

// Debounce/I_Debounce
INTERFACE I_Debounce EXTENDS I_BaseCyclic

PROPERTY P_DebounceStatus : REFERENCE TO ST_DebounceStatus
GET
END_GET
END_PROPERTY

PROPERTY P_RawSignal : BOOL
GET
END_GET
SET
END_SET
END_PROPERTY

END_INTERFACE

// EventHandling/ITFs/I_LogHandler
INTERFACE I_LogHandler EXTENDS __SYSTEM.IQueryInterface

METHOD AddToEventLog : BOOL
END_METHOD

METHOD LogDequeue
END_METHOD

METHOD MonitorPlcSystem
END_METHOD

PROPERTY P_EventLogHandlerStatus : REFERENCE TO ST_EventLogHandlerStatus
GET
END_GET
END_PROPERTY

END_INTERFACE

// EventHandling/ITFs/I_LogHandlerConfiguration
INTERFACE I_LogHandlerConfiguration EXTENDS __SYSTEM.IQueryInterface

PROPERTY P_EventLogHandlerConfiguration : REFERENCE TO ST_EventLogHandlerConfiguration
GET
END_GET
END_PROPERTY

END_INTERFACE

// EventHandling/ITFs/I_PersistentStorage
INTERFACE I_PersistentStorage EXTENDS __SYSTEM.IQueryInterface

METHOD PUBLIC AddEntry : BOOL
VAR_INPUT
	Source		: T_MaxString;
	Message 	: T_MaxString;
	Flags		: UDINT;
	PlcTaskInfo	: Global.PlcTaskSystemInfo;
	Severity 	: Global.TcEventSeverity;
	RaiseAlarm	: BOOL;
END_VAR
END_METHOD

PROPERTY P_MessagesSentThisScan : REFERENCE TO UDINT
GET
END_GET
END_PROPERTY

END_INTERFACE

// EventHandling/ITFs/I_TraceEvent
INTERFACE I_TraceEvent EXTENDS __SYSTEM.IQueryInterface

METHOD AddContext
VAR_INPUT
	Source 			: T_MaxString;
	PlcTaskInfo		: Global.PlcTaskSystemInfo;
	Flags  			: UDINT;
END_VAR
END_METHOD

METHOD SetMessage
VAR_INPUT
    Message : T_MaxString;
END_VAR
END_METHOD

METHOD SetSeverity
VAR_INPUT
    Severity : Global.TcEventSeverity;
END_VAR
END_METHOD

END_INTERFACE

// EventHandling/FB_EventLogHandler
FUNCTION_BLOCK FB_EventLogHandler EXTENDS FB_BaseCyclic IMPLEMENTS I_LogHandler, I_LogHandlerConfiguration
VAR
	EventLogHandlerConfiguration	: ST_EventLogHandlerConfiguration;
	EventLogHandlerStatus			: ST_EventLogHandlerStatus;
	TEST_EventLogHandlerStatus		: ST_EventLogHandlerStatus; //ONLY for tests
	
	LogEntry						: ST_LogEntry;
	
	// Task monitoring variables
	ForIndex				: DINT;					// Loop index for task iteration
	SafeTaskCount			: UDINT;				// Cached task count to avoid race conditions
	MaxTaskIndex			: DINT;					// Safe upper bound for task iteration

	// Debug/diagnostic variables (consider making these temporary)
	DebugSingleStep			: BOOL;					// When TRUE, process only one event per cycle
	DebugTryAddCount		: UDINT;				// Count of TryAddToEventLog calls
	DebugTryAddSuccess		: UDINT;				// Count of successful adds
	DebugTryAddFailed		: UDINT;				// Count of failed adds
END_VAR

METHOD CyclicLogic
SUPER^.CyclicLogic();

//MOVED TO _InitializeChildrenDependencies();
// Check and handle first cycle with bounds checking
// Verify INDEX_LOG_TASK is within bounds before accessing
// IF GPL_Base.INDEX_LOG_TASK >= LOWER_BOUND(GVL_System.PlcSystemInfo, 1) AND
//    GPL_Base.INDEX_LOG_TASK <= UPPER_BOUND(GVL_System.PlcSystemInfo, 1) THEN
// 
// 	GVL_System.PlcSystemInfo[GPL_Base.INDEX_LOG_TASK].FirstCycle :=
// 		TwinCAT_SystemInfoVarList._TaskInfo[Tc2_System.GETCURTASKINDEXEX()].FirstCycle;
// ELSE
// 	RETURN;
// END_IF
// 
// // Initialize on first cycle
// IF GVL_System.PlcSystemInfo[GPL_Base.INDEX_LOG_TASK].FirstCycle THEN
// 	GVL_System.RingBufferLog.Initialize();
// 	GVL_System.GlobalEventLog.Initialize();
// 	RETURN;
// END_IF

// Normal operation
MonitorPlcSystem();
LogDequeue();
END_METHOD

METHOD AddToEventLog : BOOL
IF GVL_System.iPersistentStorage = 0 THEN
	AddToEventLog	:= FALSE;
	RETURN;
END_IF

// Add entry to EventLog using local LogEntry variable
IF GVL_System.iPersistentStorage <> 0 THEN
	// AddEntry method returns TRUE on success, FALSE on failure
	AddToEventLog := GVL_System.iPersistentStorage.AddEntry(
		RaiseAlarm := LogEntry.RaiseAlarm,
		Message := LogEntry.Message,
		Severity := LogEntry.Severity,
		Source := LogEntry.InstancePath,
		PlcTaskInfo := LogEntry.TaskInfo,
		Flags := 0
	);
ELSE
	AddToEventLog := FALSE;
END_IF
END_METHOD

METHOD LogDequeue
IF GPL_Base.TRACING_ENABLED THEN
	// Always reset counters at start of each cycle
	EventLogHandlerStatus.LogCountThisScan := 0;
	IF GVL_System.iPersistentStorage <> 0 THEN
		GVL_System.iPersistentStorage.P_MessagesSentThisScan := 0;
	END_IF
	EventLogHandlerStatus.CycleStartTime := ULINT_TO_UDINT(Tc2_System.F_GetSystemTime());

	// Update buffer health metrics
	UpdateBufferHealthMetrics();

	// Update exponential backoff timer
	EventLogHandlerStatus.BackoffState.BackoffTimer(IN := EventLogHandlerStatus.BackoffState.PersistenceBlocked, PT := UDINT_TO_TIME(EventLogHandlerStatus.BackoffState.BackoffDelayMs));
	IF EventLogHandlerStatus.BackoffState.BackoffTimer.Q THEN
		EventLogHandlerStatus.BackoffState.PersistenceBlocked := FALSE;
		EventLogHandlerStatus.BackoffState.BackoffDelayMs := 0;
		// FIXED: Removed increment here - BackoffActiveCount is now incremented when backoff starts
		IF EventLogHandlerConfiguration.BaseConfiguration.LogTraceConfiguration.What.xLogToEventLogger THEN
			ADSLOGSTR(
				msgCtrlMask := ADSLOG_MSGTYPE_HINT,
				msgFmtStr := 'EventLogHandler: Backoff period complete, resuming processing',
				strArg := ''
			);
		END_IF
	END_IF;

	// Calculate dynamic processing rate based on system load
	EventLogHandlerStatus.DynamicMaxEntries := CalculateDynamicRate();

	// Check for forced buffer reset due to corruption
	IF EventLogHandlerStatus.ForceBufferReset THEN
		// Force clear the buffer state
		ADSLOGSTR(
			msgCtrlMask := ADSLOG_MSGTYPE_WARN,
			msgFmtStr := 'EventLogHandler: Forcing buffer reset due to corruption detection',
			strArg := ''
		);

		// Reset buffer by clearing all entries
		WHILE GVL_System.RingBufferLog.P_RingBufferStatus.ObjectCountInBufferPrim > 0 DO
			GVL_System.RingBufferLog.RemoveObject();
			IF GVL_System.RingBufferLog.P_ObjectWasRemoved THEN
				GVL_System.RingBufferLog.ClearStatusFlagRemoved();
				GVL_System.RingBufferLog.ClearLastRemoved();
			ELSE
				// Can't remove - force exit to prevent infinite loop
				EXIT;
			END_IF
		END_WHILE

		// Clear all tracking flags
		EventLogHandlerStatus.ForceBufferReset := FALSE;
		EventLogHandlerStatus.BufferCorruptionDetected := FALSE;
		EventLogHandlerStatus.ConsecutiveRemoveFailures := 0;
		EventLogHandlerStatus.ConsecutiveEmptyScans := 0;
	END_IF

	// Determine if we should process entries
	// Process if: buffer has items AND system has capacity AND not blocked
	EventLogHandlerStatus.ShouldProcess := (GVL_System.RingBufferLog.P_RingBufferStatus.ObjectCountInBufferPrim > 0) AND
					 (EventLogHandlerStatus.DynamicMaxEntries > 0) AND
					 NOT EventLogHandlerStatus.BackoffState.PersistenceBlocked AND
					 NOT EventLogHandlerStatus.BufferCorruptionDetected;

	IF EventLogHandlerStatus.ShouldProcess THEN
		// Debug mode: process one event at a time, but continue until buffer empty
		IF DebugSingleStep THEN
			REPEAT
				_ProcessLogEntry(ShouldExit => EventLogHandlerStatus.ExitProcessing);

				IF EventLogHandlerStatus.ExitProcessing THEN
					EventLogHandlerStatus.ExitProcessing	:= FALSE;
					EXIT; // Stop processing on failure
				END_IF;

			UNTIL (GVL_System.RingBufferLog.P_RingBufferStatus.ObjectCountInBufferPrim = 0)
			END_REPEAT
		ELSE
			// Normal mode: process multiple events per cycle up to rate limit
			REPEAT
				_ProcessLogEntry(ShouldExit => EventLogHandlerStatus.ExitProcessing);

				IF EventLogHandlerStatus.ExitProcessing THEN
					EventLogHandlerStatus.ExitProcessing	:= FALSE;
					EXIT; // Stop processing on failure
				END_IF;

			UNTIL (GVL_System.RingBufferLog.P_RingBufferStatus.ObjectCountInBufferPrim = 0) OR
				  (EventLogHandlerStatus.LogCountThisScan >= EventLogHandlerStatus.DynamicMaxEntries) OR
				  EventLogHandlerStatus.BackoffState.PersistenceBlocked
			END_REPEAT
		END_IF;
	END_IF;

	// Track consecutive empty scans for cycle break protection
	IF EventLogHandlerStatus.LogCountThisScan = 0 AND EventLogHandlerStatus.ShouldProcess THEN
		// We tried to process but got nothing done
		EventLogHandlerStatus.ConsecutiveEmptyScans := EventLogHandlerStatus.ConsecutiveEmptyScans + 1;

		// Check for excessive empty scans
		IF EventLogHandlerStatus.ConsecutiveEmptyScans >= 10 THEN
			// Force backoff to break the cycle
			EventLogHandlerStatus.BackoffState.PersistenceBlocked := TRUE;
			EventLogHandlerStatus.BackoffState.BackoffDelayMs := 5000; // 5 second forced backoff
			ADSLOGSTR(
				msgCtrlMask := ADSLOG_MSGTYPE_WARN,
				msgFmtStr := 'EventLogHandler: 10 consecutive empty scans detected - forcing 5 second backoff',
				strArg := ''
			);
			// Reset counter to prevent continuous backoff
			EventLogHandlerStatus.ConsecutiveEmptyScans := 0;
		END_IF
	ELSIF EventLogHandlerStatus.LogCountThisScan > 0 THEN
		// Successful processing - reset counter and update timestamp
		EventLogHandlerStatus.ConsecutiveEmptyScans := 0;
		EventLogHandlerStatus.LastSuccessfulProcessTime := ULINT_TO_UDINT(Tc2_System.F_GetSystemTime());
	END_IF

	// Update performance metrics
	_UpdatePerformanceMetrics(EventLogHandlerStatus.CycleStartTime);
END_IF
END_METHOD

METHOD MonitorPlcSystem
// Capture task count once to avoid race conditions
SafeTaskCount := TwinCAT_SystemInfoVarList._AppInfo.TaskCnt;

// Calculate safe upper bound - clamp against all array bounds
MaxTaskIndex := MIN(
	UDINT_TO_DINT(SafeTaskCount),
	UPPER_BOUND(GVL_System.PlcSystemInfo, 1),
	UPPER_BOUND(TwinCAT_SystemInfoVarList._TaskInfo, 1)
);

IF (LOWER_BOUND(GVL_System.PlcSystemInfo,1)+1) <= MaxTaskIndex THEN
	FOR ForIndex := (LOWER_BOUND(GVL_System.PlcSystemInfo,1)+1) TO MaxTaskIndex BY 1 DO
		// Double-check bounds before each access (defensive programming)
		IF ForIndex > UPPER_BOUND(TwinCAT_SystemInfoVarList._TaskInfo, 1) THEN
			EXIT;  // Task array has shrunk, exit safely
		END_IF
	
		IF ForIndex > UPPER_BOUND(GVL_System.PlcSystemInfo, 1) THEN
			EXIT;  // Prevent overrun
		END_IF
	
		// Copy task information
		GVL_System.PlcSystemInfo[ForIndex].CycleTimeExceeded := TwinCAT_SystemInfoVarList._TaskInfo[ForIndex].CycleTimeExceeded;
		GVL_System.PlcSystemInfo[ForIndex].RTViolation := TwinCAT_SystemInfoVarList._TaskInfo[ForIndex].RTViolation;
	
		// Calculate utilization only if cycle time is valid
		IF TwinCAT_SystemInfoVarList._TaskInfo[ForIndex].CycleTime <> 0 THEN
			GVL_System.PlcSystemInfo[ForIndex].TaskUtilizationPercentage :=
				TwinCAT_SystemInfoVarList._TaskInfo[ForIndex].LastExecTime /
				TwinCAT_SystemInfoVarList._TaskInfo[ForIndex].CycleTime;
		END_IF
	
		// FIXED: Call R_TRIG instances BEFORE checking Q output
		// Update edge detection triggers first
		GVL_System.PlcSystemInfo[ForIndex].LogCycleExceed(CLK := GVL_System.PlcSystemInfo[ForIndex].CycleTimeExceeded);
		GVL_System.PlcSystemInfo[ForIndex].LogRTViolation(CLK := GVL_System.PlcSystemInfo[ForIndex].RTViolation);
	
		// Log cycle exceed events (rising edge detection)
		IF GVL_System.PlcSystemInfo[ForIndex].LogCycleExceed.Q THEN
			ADSLOGSTR(
				msgCtrlMask := ADSLOG_MSGTYPE_ERROR,
				msgFmtStr := 'EventLogHandler: Cycle Exceed in Task %s',
				strArg := GVL_System.PlcSystemInfo[ForIndex].TaskName
			);
		END_IF

		// Log RT violation events (rising edge detection)
		IF GVL_System.PlcSystemInfo[ForIndex].LogRTViolation.Q THEN
			ADSLOGSTR(
				msgCtrlMask := ADSLOG_MSGTYPE_ERROR,
				msgFmtStr := 'EventLogHandler: RT Violation in Task %s',
				strArg := GVL_System.PlcSystemInfo[ForIndex].TaskName
			);
		END_IF
	END_FOR
END_IF
END_METHOD

PROPERTY P_EventLogHandlerStatus : REFERENCE TO ST_EventLogHandlerStatus
GET
IF EventLogHandlerConfiguration.BaseConfiguration.InSimulation THEN
	P_EventLogHandlerStatus	REF= TEST_EventLogHandlerStatus;
ELSE
	P_EventLogHandlerStatus REF= EventLogHandlerStatus;
END_IF
END_GET
END_PROPERTY

PROPERTY P_EventLogHandlerConfiguration : REFERENCE TO ST_EventLogHandlerConfiguration
GET
P_EventLogHandlerConfiguration REF= EventLogHandlerConfiguration;
END_GET
END_PROPERTY

METHOD PROTECTED _InitializeChildrenDependencies : BOOL
GVL_System.RingBufferLog.Initialize();
GVL_System.GlobalEventLog.Initialize();

_InitializeChildrenDependencies := TRUE;
END_METHOD

METHOD PROTECTED _InitializeReferences : BOOL
//Order is important!
BaseConfiguration.InstancePath 	REF= InstancePath;

// Note: Removed cyclic trace message - _InitializeReferences is called repeatedly during init attempts
// If you created new data structures, they may not have valid pointer references

EventLogHandlerConfiguration.BaseConfiguration	REF= SUPER^.BaseConfiguration;

EventLogHandlerStatus.BaseStatus				REF= SUPER^.BaseStatus;

TEST_EventLogHandlerStatus.BaseStatus			REF= SUPER^.BaseStatus;

_InitializeReferences 			:= TRUE; // apply at end of all reference initialization
END_METHOD

METHOD PROTECTED _ProcessLogEntry : BOOL
VAR_OUTPUT
	ShouldExit	: BOOL;		// TRUE if processing should stop (failure occurred)
END_VAR
// Initialize return values
_ProcessLogEntry := FALSE;
ShouldExit := FALSE;

// Remove entry from ring buffer
GVL_System.RingBufferLog.RemoveObject();

IF GVL_System.RingBufferLog.P_ObjectWasRemoved THEN
	LogEntry := GVL_System.RingBufferLog.P_LastObjectRemoved;
	GVL_System.RingBufferLog.ClearStatusFlagRemoved();

	// Reset consecutive failure counter on successful remove
	EventLogHandlerStatus.ConsecutiveRemoveFailures := 0;

	// Track retry count for monitoring
	EventLogHandlerStatus.CurrentEntryRetryCount := LogEntry.RetryCount;

	EventLogHandlerStatus.PersistenceSuccess := AddToEventLog();
	// Attempt to add to EventLog with error handling
	DebugTryAddCount := DebugTryAddCount + 1;

	IF EventLogHandlerStatus.PersistenceSuccess THEN
		DebugTryAddSuccess := DebugTryAddSuccess + 1;
		// Reset failure count on successful persistence
		EventLogHandlerStatus.BackoffState.PersistenceFailureCount := 0;
		EventLogHandlerStatus.BackoffState.PersistenceBlocked := FALSE; // Clear any active backoff
		EventLogHandlerStatus.CurrentEntryRetryCount := 0;
		EventLogHandlerStatus.LogCountThisScan := EventLogHandlerStatus.LogCountThisScan + 1;
		// FIXED: Don't increment EntriesProcessedThisCycle here - it gets set from LogCountThisScan later
		EventLogHandlerStatus.LoggingMetrics.TotalEntriesProcessed := EventLogHandlerStatus.LoggingMetrics.TotalEntriesProcessed + 1;

		// Update severity-specific counters
		_UpdateSeverityMetrics();

		_ProcessLogEntry := TRUE;
	ELSE
		DebugTryAddFailed := DebugTryAddFailed + 1;

		// Increment retry count for this entry
		LogEntry.RetryCount := LogEntry.RetryCount + 1;

		IF EventLogHandlerConfiguration.BaseConfiguration.LogTraceConfiguration.What.xLogToEventLogger THEN
			ADSLOGSTR(
				msgCtrlMask := ADSLOG_MSGTYPE_WARN,
				msgFmtStr := 'EventLogHandler: Persistence failed for entry, retry count: %s',
				strArg := UINT_TO_STRING(LogEntry.RetryCount)
			);
		END_IF

		// Check if max retries exceeded
		IF LogEntry.RetryCount >= EventLogHandlerConfiguration.MaxRetryAttemptsPerEntry THEN
			// Discard entry after max retries - log critical error
			ADSLOGSTR(
				msgCtrlMask := ADSLOG_MSGTYPE_ERROR,
				msgFmtStr := 'EventLogHandler: Max retries exceeded, discarding log entry',
				strArg := ''
			);
			EventLogHandlerStatus.LoggingMetrics.PersistenceFailureCount := EventLogHandlerStatus.LoggingMetrics.PersistenceFailureCount + 1;
		ELSE
			// On failure: Only re-add entry if we're not entering backoff
			// This prevents the buffer from filling with entries that will immediately fail again
			IF EventLogHandlerStatus.BackoffState.PersistenceFailureCount < 3 THEN
				// Still within reasonable retry attempts - re-add to buffer
				IF GVL_System.iBuffer <> 0 THEN
					GVL_System.iBuffer.AddObject(RefObject := LogEntry);

					// Check if the re-add succeeded
					IF GVL_System.RingBufferLog.P_ObjectWasAdded THEN
						IF EventLogHandlerConfiguration.BaseConfiguration.LogTraceConfiguration.What.xLogToEventLogger THEN
							ADSLOGSTR(
								msgCtrlMask := ADSLOG_MSGTYPE_HINT,
								msgFmtStr := 'EventLogHandler: Re-added entry to buffer for retry',
								strArg := ''
							);
						END_IF
						GVL_System.RingBufferLog.ClearStatusFlagAdded();
					ELSE
						// Re-add failed - entry will be lost
						ADSLOGSTR(
							msgCtrlMask := ADSLOG_MSGTYPE_ERROR,
							msgFmtStr := 'EventLogHandler: Failed to re-add entry to buffer - entry lost',
							strArg := ''
						);
						EventLogHandlerStatus.LoggingMetrics.PersistenceFailureCount := EventLogHandlerStatus.LoggingMetrics.PersistenceFailureCount + 1;
					END_IF
				ELSE
					ADSLOGSTR(
						msgCtrlMask := ADSLOG_MSGTYPE_ERROR,
						msgFmtStr := 'EventLogHandler: iBuffer interface is NULL, cannot re-add entry for retry',
						strArg := ''
					);
				END_IF
			ELSE
				// Too many consecutive failures - discard entry to prevent ping-pong
				ADSLOGSTR(
					msgCtrlMask := ADSLOG_MSGTYPE_WARN,
					msgFmtStr := 'EventLogHandler: Discarding entry due to repeated failures - entering backoff',
					strArg := ''
				);
				EventLogHandlerStatus.LoggingMetrics.PersistenceFailureCount := EventLogHandlerStatus.LoggingMetrics.PersistenceFailureCount + 1;
			END_IF
		END_IF

		// Handle persistence failure with exponential backoff
		HandlePersistenceFailure();
		ShouldExit := TRUE;
	END_IF;

	// Always clear the last removed entry to keep the buffer moving
	GVL_System.iBuffer.ClearLastRemoved();
ELSE
	// RemoveObject was called but nothing was removed - buffer may be empty or corrupted
	DebugTryAddFailed := DebugTryAddFailed + 1;
	EventLogHandlerStatus.ConsecutiveRemoveFailures := EventLogHandlerStatus.ConsecutiveRemoveFailures + 1;

	// Check if we've hit the failure threshold
	IF EventLogHandlerStatus.ConsecutiveRemoveFailures >= 5 THEN
		// Buffer is likely corrupted - force a reset
		EventLogHandlerStatus.BufferCorruptionDetected := TRUE;
		EventLogHandlerStatus.ForceBufferReset := TRUE;
		ADSLOGSTR(
			msgCtrlMask := ADSLOG_MSGTYPE_ERROR,
			msgFmtStr := 'EventLogHandler: Buffer corruption detected after 5 consecutive RemoveObject failures - forcing reset',
			strArg := ''
		);
	ELSE
		ADSLOGSTR(
			msgCtrlMask := ADSLOG_MSGTYPE_ERROR,
			msgFmtStr := 'EventLogHandler: LogDequeue RemoveObject failed - buffer may be empty or corrupted',
			strArg := ''
		);
	END_IF
	ShouldExit := TRUE;
END_IF;
END_METHOD

METHOD PROTECTED _UpdatePerformanceMetrics
VAR_INPUT
	CycleStartTime		: UDINT;
END_VAR
VAR
	CycleEndTime		: UDINT;		// End time for this processing cycle
	ProcessingTimeMs	: UDINT;		// Time taken to process entries
END_VAR
// Calculate cycle utilization and processing time
CycleEndTime := ULINT_TO_UDINT(Tc2_System.F_GetSystemTime());
ProcessingTimeMs := CycleEndTime - CycleStartTime;

// Update current cycle metrics (utilization already updated by MonitorPlcSystem)
EventLogHandlerStatus.LoggingMetrics.CycleUtilizationPercentage := GVL_System.PlcSystemInfo[GPL_BASE.INDEX_LOG_TASK].TaskUtilizationPercentage * GC_Base.PercentageMultiplier;
EventLogHandlerStatus.LoggingMetrics.EntriesProcessedThisCycle := EventLogHandlerStatus.LogCountThisScan;

// Track peak processing time
IF ProcessingTimeMs > EventLogHandlerStatus.LoggingMetrics.PeakProcessingTimeMs THEN
    EventLogHandlerStatus.LoggingMetrics.PeakProcessingTimeMs := ProcessingTimeMs;
END_IF;

// Update rolling average processing time (simple moving average)
EventLogHandlerStatus.LoggingMetrics.AverageProcessingTimeMs := (EventLogHandlerStatus.LoggingMetrics.AverageProcessingTimeMs * EventLogHandlerConfiguration.RollingAvgWeightPrevious) + (UDINT_TO_REAL(ProcessingTimeMs) * EventLogHandlerConfiguration.RollingAvgWeightCurrent);

// FIXED: Calculate entries per second based on actual measured processing time (convert ms to seconds)
IF ProcessingTimeMs > 0 THEN
    EventLogHandlerStatus.LoggingMetrics.EntriesProcessedPerSecond := (UDINT_TO_REAL(EventLogHandlerStatus.LogCountThisScan) / (UDINT_TO_REAL(ProcessingTimeMs) / GC_Base.MillisecondsPerSecond));
ELSE
    EventLogHandlerStatus.LoggingMetrics.EntriesProcessedPerSecond := 0.0;
END_IF;

// Calculate overall system health score (0-100%)
// Based on: low utilization, low buffer usage, no failures, no cycle exceeds (from MonitorPlcSystem)
// FIXED: SEL logic - SEL(G,A,B) returns B when G=TRUE, A when FALSE
EventLogHandlerStatus.LoggingMetrics.SystemHealthScore :=
    GC_Base.PercentageMultiplier -
    (EventLogHandlerStatus.LoggingMetrics.CycleUtilizationPercentage * EventLogHandlerConfiguration.HealthScoreUtilizationWeight) -
    (EventLogHandlerStatus.LoggingMetrics.BufferUtilizationPercentage * EventLogHandlerConfiguration.HealthScoreBufferWeight) -
    (SEL(EventLogHandlerStatus.BackoffState.PersistenceFailureCount > 0, EventLogHandlerConfiguration.HealthScorePersistencePenalty, 0.0)) -  // Subtract penalty when failures exist
    (SEL(GVL_System.PlcSystemInfo[GPL_BASE.INDEX_LOG_TASK].CycleTimeExceeded, 0.0, EventLogHandlerConfiguration.HealthScoreCycleExceedPenalty));  // Subtract penalty when cycle exceeded

EventLogHandlerStatus.LoggingMetrics.SystemHealthScore := MAX(0.0, EventLogHandlerStatus.LoggingMetrics.SystemHealthScore);
END_METHOD

METHOD PROTECTED _UpdateSeverityMetrics
// Update severity-specific counters based on last processed entry
CASE LogEntry.Severity OF
    Global.TcEventSeverity.Critical:
        EventLogHandlerStatus.LoggingMetrics.CriticalEntriesProcessed := EventLogHandlerStatus.LoggingMetrics.CriticalEntriesProcessed + 1;
    Global.TcEventSeverity.Error:
        EventLogHandlerStatus.LoggingMetrics.ErrorEntriesProcessed := EventLogHandlerStatus.LoggingMetrics.ErrorEntriesProcessed + 1;
    Global.TcEventSeverity.Warning:
        EventLogHandlerStatus.LoggingMetrics.WarningEntriesProcessed := EventLogHandlerStatus.LoggingMetrics.WarningEntriesProcessed + 1;
    Global.TcEventSeverity.Info, Global.TcEventSeverity.Verbose:
        EventLogHandlerStatus.LoggingMetrics.InfoEntriesProcessed := EventLogHandlerStatus.LoggingMetrics.InfoEntriesProcessed + 1;
END_CASE;
END_METHOD

METHOD CalculateDynamicRate : UINT
VAR
	BufferUtilizationPercentage	: REAL;		// Local calculation of buffer usage
END_VAR
// Calculate buffer utilization
BufferUtilizationPercentage := UDINT_TO_REAL(GVL_System.RingBufferLog.P_RingBufferStatus.ObjectCountInBufferPrim) /
                               UDINT_TO_REAL(GVL_System.RingBufferLog.P_RingBufferStatus.BufferCapacity) * GC_Base.PercentageMultiplier;

// Start with base rate
EventLogHandlerStatus.DynamicMaxEntries := UDINT_TO_UINT(GPL_Base.MAX_LOG_ENTRIES_PER_SCAN);

// Adjust based on task utilization
IF GVL_System.PlcSystemInfo[GPL_BASE.INDEX_LOG_TASK].TaskUtilizationPercentage > GPL_BASE.LOG_CYCLE_EXCEED_MAX_THRESHOLD THEN
    // High load: reduce to quarter rate
    EventLogHandlerStatus.DynamicMaxEntries := UDINT_TO_UINT(GPL_Base.MAX_LOG_ENTRIES_PER_SCAN / EventLogHandlerConfiguration.RateDivisorHighLoad);
ELSIF GVL_System.PlcSystemInfo[GPL_BASE.INDEX_LOG_TASK].TaskUtilizationPercentage > EventLogHandlerConfiguration.TaskUtilModerateThreshold THEN
    // Moderate load: half rate
    EventLogHandlerStatus.DynamicMaxEntries := UDINT_TO_UINT(GPL_Base.MAX_LOG_ENTRIES_PER_SCAN / EventLogHandlerConfiguration.RateDivisorModerateLoad);
ELSIF GVL_System.PlcSystemInfo[GPL_BASE.INDEX_LOG_TASK].TaskUtilizationPercentage < EventLogHandlerConfiguration.TaskUtilLowThreshold THEN
    // Low load: increase rate if buffer is filling up
    IF BufferUtilizationPercentage >= EventLogHandlerConfiguration.BufferThresholdIncrease THEN
        EventLogHandlerStatus.DynamicMaxEntries := UDINT_TO_UINT(GPL_Base.MAX_LOG_ENTRIES_PER_SCAN * EventLogHandlerConfiguration.RateMultiplierLowLoad);
    END_IF;
END_IF;

// Emergency mode: if buffer is nearly full, prioritize draining
IF BufferUtilizationPercentage >= EventLogHandlerConfiguration.BufferThresholdEmergency THEN
    EventLogHandlerStatus.DynamicMaxEntries := UDINT_TO_UINT(GPL_Base.MAX_LOG_ENTRIES_PER_SCAN * EventLogHandlerConfiguration.EmergencyRateMultiplier);
ELSIF BufferUtilizationPercentage >= EventLogHandlerConfiguration.BufferThresholdHigh THEN
    EventLogHandlerStatus.DynamicMaxEntries := MIN(UDINT_TO_UINT(UINT_TO_UDINT(EventLogHandlerStatus.DynamicMaxEntries) * EventLogHandlerConfiguration.HighBufferRateMultiplier), UDINT_TO_UINT(GPL_Base.MAX_LOG_ENTRIES_PER_SCAN * EventLogHandlerConfiguration.HighBufferRateMultiplier));
END_IF;

// Ensure we don't exceed absolute maximum
EventLogHandlerStatus.DynamicMaxEntries := MIN(EventLogHandlerStatus.DynamicMaxEntries, EventLogHandlerConfiguration.MaxEntriesPerScanAbsolute);

// Return calculated value
CalculateDynamicRate := EventLogHandlerStatus.DynamicMaxEntries;
END_METHOD

METHOD HandlePersistenceFailure
// Implement exponential backoff on persistence failures
EventLogHandlerStatus.BackoffState.PersistenceFailureCount := EventLogHandlerStatus.BackoffState.PersistenceFailureCount + 1;
EventLogHandlerStatus.LoggingMetrics.PersistenceFailureCount := EventLogHandlerStatus.LoggingMetrics.PersistenceFailureCount + 1;

// Calculate exponential backoff delay: InitialDelay * Multiplier^(failures-1), max MaxDelay
IF EventLogHandlerStatus.BackoffState.PersistenceFailureCount = 1 THEN
    EventLogHandlerStatus.BackoffState.BackoffDelayMs := EventLogHandlerConfiguration.BackoffInitialDelayMs;
ELSIF EventLogHandlerStatus.BackoffState.PersistenceFailureCount = 2 THEN
    EventLogHandlerStatus.BackoffState.BackoffDelayMs := REAL_TO_UDINT(EventLogHandlerConfiguration.BackoffInitialDelayMs * EventLogHandlerConfiguration.BackoffMultiplier);
ELSIF EventLogHandlerStatus.BackoffState.PersistenceFailureCount = 3 THEN
    EventLogHandlerStatus.BackoffState.BackoffDelayMs := REAL_TO_UDINT(EventLogHandlerConfiguration.BackoffInitialDelayMs * EventLogHandlerConfiguration.BackoffMultiplier * EventLogHandlerConfiguration.BackoffMultiplier);
ELSIF EventLogHandlerStatus.BackoffState.PersistenceFailureCount = 4 THEN
    EventLogHandlerStatus.BackoffState.BackoffDelayMs := REAL_TO_UDINT(EventLogHandlerConfiguration.BackoffInitialDelayMs * EventLogHandlerConfiguration.BackoffMultiplier * EventLogHandlerConfiguration.BackoffMultiplier * EventLogHandlerConfiguration.BackoffMultiplier);
ELSIF EventLogHandlerStatus.BackoffState.PersistenceFailureCount = 5 THEN
    EventLogHandlerStatus.BackoffState.BackoffDelayMs := REAL_TO_UDINT(EventLogHandlerConfiguration.BackoffInitialDelayMs * EventLogHandlerConfiguration.BackoffMultiplier * EventLogHandlerConfiguration.BackoffMultiplier * EventLogHandlerConfiguration.BackoffMultiplier * EventLogHandlerConfiguration.BackoffMultiplier);
ELSIF EventLogHandlerStatus.BackoffState.PersistenceFailureCount = 6 THEN
    EventLogHandlerStatus.BackoffState.BackoffDelayMs := REAL_TO_UDINT(EventLogHandlerConfiguration.BackoffInitialDelayMs * EventLogHandlerConfiguration.BackoffMultiplier * EventLogHandlerConfiguration.BackoffMultiplier * EventLogHandlerConfiguration.BackoffMultiplier * EventLogHandlerConfiguration.BackoffMultiplier * EventLogHandlerConfiguration.BackoffMultiplier);
ELSE
    EventLogHandlerStatus.BackoffState.BackoffDelayMs := EventLogHandlerConfiguration.BackoffMaxDelayMs; // Cap at max delay
END_IF;

// Activate backoff
EventLogHandlerStatus.BackoffState.PersistenceBlocked := TRUE;
EventLogHandlerStatus.LoggingMetrics.CurrentBackoffDelayMs := EventLogHandlerStatus.BackoffState.BackoffDelayMs;
EventLogHandlerStatus.LoggingMetrics.TotalBackoffTimeMs := EventLogHandlerStatus.LoggingMetrics.TotalBackoffTimeMs + EventLogHandlerStatus.BackoffState.BackoffDelayMs;
// FIXED: Increment BackoffActivations when backoff is activated, not when it exits
EventLogHandlerStatus.LoggingMetrics.BackoffActiveCount := EventLogHandlerStatus.LoggingMetrics.BackoffActiveCount + 1;
END_METHOD

METHOD UpdateBufferHealthMetrics
VAR
	BufferUtilizationPercentage	: REAL;		// Local calculation of buffer usage
END_VAR
// Calculate current buffer utilization percentage
BufferUtilizationPercentage := UDINT_TO_REAL(GVL_System.RingBufferLog.P_RingBufferStatus.ObjectCountInBufferPrim) /
                               UDINT_TO_REAL(GVL_System.RingBufferLog.P_RingBufferStatus.BufferCapacity) * GC_Base.PercentageMultiplier;

// Update metrics structure
EventLogHandlerStatus.LoggingMetrics.BufferUtilizationPercentage := BufferUtilizationPercentage;

// Track peak utilization
IF BufferUtilizationPercentage > EventLogHandlerStatus.LoggingMetrics.MaxBufferUtilizationReached THEN
    EventLogHandlerStatus.LoggingMetrics.MaxBufferUtilizationReached := BufferUtilizationPercentage;
END_IF;

// FIXED: Count buffer overflows using edge detection (only increment on rising edge)
EventLogHandlerStatus.BufferOverflowTrigger(CLK := GVL_System.RingBufferLog.P_RingBufferStatus.BufferIsFullPrim);
IF EventLogHandlerStatus.BufferOverflowTrigger.Q THEN
    EventLogHandlerStatus.LoggingMetrics.BufferOverflowCount := EventLogHandlerStatus.LoggingMetrics.BufferOverflowCount + 1;
END_IF;
END_METHOD

END_FUNCTION_BLOCK

// EventHandling/FB_PersistentEventLog
{attribute 'no_explicit_call' := 'do not call this POU directly'}
FUNCTION_BLOCK FB_PersistentEventLog EXTENDS FB_BaseStatic IMPLEMENTS I_PersistentStorage
VAR
	PersistentStorageStatus		: ST_PersistentStorageStatus;
	
	//Configuration
	TracingAllowed				: BOOL := TRUE;
	
	UniversalMessage			: FB_UniversalMessage;
	UniversalAlarm				: FB_UniversalAlarm;
END_VAR

METHOD PROTECTED _InitializeChildrenDependencies : BOOL
// Initialize child components
IF NOT UniversalMessage.P_BaseStatus.Initialized THEN
	_InitializeChildrenDependencies := UniversalMessage.Initialize();
END_IF

IF NOT UniversalAlarm.P_BaseStatus.Initialized THEN
	_InitializeChildrenDependencies := UniversalAlarm.Initialize();
END_IF

_InitializeChildrenDependencies := UniversalMessage.P_BaseStatus.Initialized AND UniversalAlarm.P_BaseStatus.Initialized;  // All children initialized successfully
END_METHOD

METHOD PROTECTED _InitializeReferences : BOOL
//Order is important!
BaseConfiguration.InstancePath 	REF= InstancePath;

PersistentStorageStatus.BaseStatus	REF= SUPER^.BaseStatus;

IF BaseConfiguration.LogTraceConfiguration.When = E_LogTraceWhen.xRunOnInitOnly AND_THEN
   BaseConfiguration.LogTraceConfiguration.What.xLogToEventLogger THEN
	ADSLOGSTR(
		msgCtrlMask := ADSLOG_MSGTYPE_WARN,
		msgFmtStr := 'PersistentEventLog: If you created new data structures, they may not have valid pointer references; Check %s',
		strArg := __POUNAME()
	);
END_IF

_InitializeReferences 			:= TRUE; // apply at end of all reference initialization
END_METHOD

METHOD PUBLIC AddEntry : BOOL
VAR_INPUT
	Source		: T_MaxString;
	Message 	: T_MaxString;
	Flags		: UDINT;
	PlcTaskInfo	: Global.PlcTaskSystemInfo;
	Severity 	: Global.TcEventSeverity;
	RaiseAlarm	: BOOL;
END_VAR
// Default to success - only set to FALSE on actual failure
AddEntry := TRUE;

IF NOT SUPER^.BaseStatus.Initialized THEN
	IF BaseConfiguration.LogTraceConfiguration.What.xLogToEventLogger AND NOT PersistentStorageStatus.NotInitializedMessageShown THEN
		ADSLOGSTR(
			msgCtrlMask := ADSLOG_MSGTYPE_WARN,
			msgFmtStr := 'PersistentEventLog not initialized, will initialize on next scan',
			strArg := ''
		);
		PersistentStorageStatus.NotInitializedMessageShown := TRUE;
	END_IF

	// Try to initialize
	IF NOT Initialize() THEN
		// Log initialization failure (use ADSLOGSTR to bypass the logging system)
		ADSLOGSTR(
			msgCtrlMask := ADSLOG_MSGTYPE_ERROR,
			msgFmtStr := 'PersistentEventLog initialization failed - check child component initialization',
			strArg := ''
		);
	END_IF

	RETURN;  // Return TRUE - initialization will be retried next scan
END_IF

IF NOT TracingAllowed THEN
	RETURN;  // Return TRUE - tracing is disabled, not a failure
END_IF

IF NOT GPL_Base.ALLOW_DUPLICATE_SEQUENTIAL_MESSAGES THEN
	// Only check for duplicates if we've sent at least one message (LastUniqueMessageTime > 0)
	// This prevents false matches against initial empty string state
	IF PersistentStorageStatus.LastUniqueMessageTime > 0 AND
	   (Source = PersistentStorageStatus.Previous_AddEntrySource) AND (Message = PersistentStorageStatus.Previous_AddEntryMessage) AND (Flags = PersistentStorageStatus.Previous_AddEntryFlags) THEN
		// Increment duplicate suppression counter
		PersistentStorageStatus.DuplicateSuppressionCount := PersistentStorageStatus.DuplicateSuppressionCount + 1;

		// Check if we should allow this duplicate through based on count or time (5 seconds)
		IF PersistentStorageStatus.DuplicateSuppressionCount >= PersistentStorageStatus.ConsecutiveDuplicateLimit OR
		   (Tc2_System.F_GetSystemTime() - PersistentStorageStatus.LastUniqueMessageTime) > 50000000 THEN  // 5 seconds in 100ns ticks
			// Too many consecutive duplicates suppressed OR too much time passed - allow this one through and reset
			IF BaseConfiguration.LogTraceConfiguration.What.xLogToEventLogger THEN
				ADSLOGSTR(
					msgCtrlMask := ADSLOG_MSGTYPE_WARN,
					msgFmtStr := 'PersistentEventLog: Forcing duplicate through after %d suppressions or timeout',
					strArg := UINT_TO_STRING(PersistentStorageStatus.DuplicateSuppressionCount)
				);
			END_IF
			PersistentStorageStatus.DuplicateSuppressionCount := 0;
			// Clear the previous entry to allow fresh duplicate detection after this one
			MEMSET(ADR(PersistentStorageStatus.Previous_AddEntrySource), 0, SIZEOF(T_MaxString));
			MEMSET(ADR(PersistentStorageStatus.Previous_AddEntryMessage), 0, SIZEOF(T_MaxString));
			// Continue to send the message
		ELSE
			// Suppress this duplicate
			RETURN;  // Return TRUE - duplicate suppression is not a failure
		END_IF
	ELSE
		// Not a duplicate - reset the suppression counter
		PersistentStorageStatus.DuplicateSuppressionCount := 0;
	END_IF
ELSE
	// Duplicate suppression is disabled - reset counter
	PersistentStorageStatus.DuplicateSuppressionCount := 0;
END_IF

// Try to send the message
AddEntry	:= FALSE;  // Will be set to TRUE if send succeeds
IF PersistentStorageStatus.MessagesSentThisScan < GPL_Base.MAX_LOG_ENTRIES_PER_SCAN THEN
	IF RaiseAlarm THEN
		// Use alarm interface with dynamic severity
		UniversalAlarm.SetSeverity(Severity);
		UniversalAlarm.SetMessage(Message);
		UniversalAlarm.AddContext(PlcTaskInfo := PlcTaskInfo, Source := Source, Flags := 0);
		AddEntry := SUCCEEDED(hr := UniversalAlarm.Raise());
	ELSE
		// Use message interface with dynamic severity
		UniversalMessage.SetSeverity(Severity);
		UniversalMessage.SetMessage(Message);
		UniversalMessage.AddContext(PlcTaskInfo := PlcTaskInfo, Source := Source, Flags := 0);
		AddEntry := SUCCEEDED(hr := UniversalMessage.Send());
	END_IF

	// Only update tracking and handle results if we actually tried to send
	IF AddEntry THEN
		PersistentStorageStatus.MessagesSentThisScan := PersistentStorageStatus.MessagesSentThisScan + 1;
		// Update previous entry tracking only when successfully sent
		MEMSET(ADR(PersistentStorageStatus.Previous_AddEntrySource), 0, SIZEOF(T_MaxString));
		MEMSET(ADR(PersistentStorageStatus.Previous_AddEntryMessage), 0, SIZEOF(T_MaxString));
		PersistentStorageStatus.Previous_AddEntrySource	 := Source;
		PersistentStorageStatus.Previous_AddEntryMessage := Message;
		PersistentStorageStatus.Previous_AddEntryFlags	 := Flags;
		PersistentStorageStatus.LastUniqueMessageTime := Tc2_System.F_GetSystemTime();  // Update timestamp for duplicate timeout tracking
	ELSE
		IF BaseConfiguration.LogTraceConfiguration.What.xLogToEventLogger THEN
			ADSLOGSTR(
				msgCtrlMask := ADSLOG_MSGTYPE_ERROR,
				msgFmtStr := 'PersistentEventLog: Event Send to LoggedEvents.db Failed: %s',
				strArg := Message
			);
		END_IF
	END_IF
ELSE
	// Scan limit reached
	IF BaseConfiguration.LogTraceConfiguration.What.xLogToEventLogger THEN
		ADSLOGSTR(
			msgCtrlMask := ADSLOG_MSGTYPE_WARN,
			msgFmtStr := 'PersistentEventLog: Max log entries per scan reached, skipping message',
			strArg := ''
		);
	END_IF
END_IF
END_METHOD

PROPERTY P_MessagesSentThisScan : REFERENCE TO UDINT
GET
P_MessagesSentThisScan REF= PersistentStorageStatus.MessagesSentThisScan;
END_GET
END_PROPERTY

END_FUNCTION_BLOCK

// EventHandling/FB_UniversalMessage
{attribute 'no_explicit_call' := 'do not call this POU directly'}
FUNCTION_BLOCK FB_UniversalMessage EXTENDS FB_TraceEvent
VAR
    fbMessage       : Tc3_EventLogger.FB_TcMessage;
    CurrentSeverity : Global.TcEventSeverity;
END_VAR

METHOD AddContext
VAR_INPUT
	Source 			: T_MaxString;
	PlcTaskInfo		: Global.PlcTaskSystemInfo;
	Flags  			: UDINT;
END_VAR
SUPER^.AddContext(PlcTaskInfo := PlcTaskInfo, Source := Source, Flags := Flags);

IF fbMessage.ipArguments <> 0 THEN
	fbMessage.ipArguments.AddString(TimeFormatter.sOut);	 // DC Timestamp string
	fbMessage.ipArguments.AddString(Source);				 // POU calling the Trace() function -- this should come automatically
	fbMessage.ipArguments.AddString(PlcTaskInfo.TaskName);	 // Task which called the POU last
	fbMessage.ipArguments.AddUDInt(PlcTaskInfo.CycleCount); 	// Cycle count of above task
	fbMessage.ipArguments.AddUDInt(Flags);					 // General-use flags (application dependent)
END_IF
END_METHOD

METHOD Send : HRESULT
VAR_INPUT
	nTimeStamp : ULINT := 0;
END_VAR
Send := fbMessage.Send(nTimeStamp);
END_METHOD

METHOD SetMessage
VAR_INPUT
    Message : T_MaxString;
END_VAR
fbMessage.ipArguments.Clear().AddString(Message);
END_METHOD

METHOD SetSeverity
VAR_INPUT
    Severity : Global.TcEventSeverity;
END_VAR
// Only recreate if severity changed
IF CurrentSeverity <> Severity THEN
    CurrentSeverity := Severity;
    
    CASE Severity OF
        Global.TcEventSeverity.Verbose,
        Global.TcEventSeverity.Info:
            fbMessage.CreateEx(TC_EVENTS.PhotaraEventClass.Info, 0);
        Global.TcEventSeverity.Warning:
            fbMessage.CreateEx(TC_EVENTS.PhotaraEventClass.Warning, 0);
        Global.TcEventSeverity.Error:
            fbMessage.CreateEx(TC_EVENTS.PhotaraEventClass.Error, 0);
//         Global.TcEventSeverity.Critical:
//             fbMessage.CreateEx(TC_EVENTS.PhotaraEventClass.Critical, 0);
        ELSE
            fbMessage.CreateEx(TC_EVENTS.PhotaraEventClass.Info, 0);
    END_CASE
END_IF
END_METHOD

END_FUNCTION_BLOCK

// EventHandling/FB_TraceEvent
FUNCTION_BLOCK ABSTRACT FB_TraceEvent EXTENDS FB_BaseStatic IMPLEMENTS I_TraceEvent
VAR
	CurrentDCTime 			: Tc2_EtherCAT.DCTIMESTRUCT;
	DCTime100Nsec 			: WORD;
	TimeFormatter			: Tc2_Utilities.FB_FormatString;
END_VAR

METHOD AddContext
VAR_INPUT
	Source 			: T_MaxString;
	PlcTaskInfo		: Global.PlcTaskSystemInfo;
	Flags  			: UDINT;
END_VAR
// Collect DC timestamp info and properly format string
CurrentDCTime := DCTIME64_TO_DCTIMESTRUCT(F_GetActualDcTime64());
DCTime100Nsec := CurrentDCTime.wNanoseconds / 100;
TimeFormatter(sFormat := '%2.2d:%2.2d:%2.2d.%3.3d%3.3d%1.1d',
			  arg1	  := F_WORD(CurrentDCTime.wHour),
			  arg2	  := F_WORD(CurrentDCTime.wMinute),
			  arg3	  := F_WORD(CurrentDCTime.wSecond),
			  arg4	  := F_WORD(CurrentDCTime.wMilliseconds),
			  arg5	  := F_WORD(CurrentDCTime.wMicroseconds),
			  arg6	  := F_WORD(DCTime100Nsec));
END_METHOD

{warning 'Add method implementation '}
METHOD SetMessage
VAR_INPUT
	Message	: T_MaxString;
END_VAR
END_METHOD

{warning 'Add method implementation '}
METHOD SetSeverity
VAR_INPUT
	Severity	: Global.TcEventSeverity;
END_VAR
END_METHOD

END_FUNCTION_BLOCK

// EventHandling/FB_UniversalAlarm
{attribute 'no_explicit_call' := 'do not call this POU directly'}
FUNCTION_BLOCK FB_UniversalAlarm EXTENDS FB_TraceEvent
VAR
    fbAlarm         : Tc3_EventLogger.FB_TcAlarm;
    CurrentSeverity : Global.TcEventSeverity;
END_VAR

METHOD AddContext
VAR_INPUT
	Source 			: T_MaxString;
	PlcTaskInfo		: Global.PlcTaskSystemInfo;
	Flags  			: UDINT;
END_VAR
SUPER^.AddContext(PlcTaskInfo := PlcTaskInfo, Source := Source, Flags := Flags);

IF fbAlarm.ipArguments <> 0 THEN 
	fbAlarm.ipArguments.AddString(TimeFormatter.sOut);	 // DC Timestamp string
	fbAlarm.ipArguments.AddString(Source);				 // POU calling the Trace() function -- this should come automatically
	fbAlarm.ipArguments.AddString(PlcTaskInfo.TaskName);	 // Task which called the POU last
	fbAlarm.ipArguments.AddUDInt(PlcTaskInfo.CycleCount); 	// Cycle count of above task
	fbAlarm.ipArguments.AddUDInt(Flags);					 // General-use flags (application dependent)
END_IF
END_METHOD

METHOD Clear : HRESULT
Clear := fbAlarm.Clear();
END_METHOD

METHOD Confirm : HRESULT
Confirm := fbAlarm.Confirm();
END_METHOD

METHOD Raise : HRESULT
VAR_INPUT
	nTimeStamp : ULINT := 0;
END_VAR
Raise := fbAlarm.Raise(nTimeStamp);
END_METHOD

METHOD SetMessage
VAR_INPUT
    Message : T_MaxString;
END_VAR
fbAlarm.ipArguments.Clear().AddString(Message);
END_METHOD

METHOD SetSeverity
VAR_INPUT
    Severity : Global.TcEventSeverity;
END_VAR
// Only recreate if severity changed
IF CurrentSeverity <> Severity THEN
    CurrentSeverity := Severity;
    
    CASE Severity OF
//         Global.TcEventSeverity.Error:
//             fbAlarm.CreateEx(TC_EVENTS.PhotaraEventClass.Alarm_ErrorWithConditonRaised, 0);
        Global.TcEventSeverity.Critical:
            fbAlarm.CreateEx(TC_EVENTS.PhotaraEventClass.Alarm_CriticalWithConditionRaised, 0);
        ELSE
            // Default to error alarm for other severities
            fbAlarm.CreateEx(TC_EVENTS.PhotaraEventClass.Alarm_CriticalWithConditionRaised, 0);
    END_CASE
END_IF
END_METHOD

END_FUNCTION_BLOCK

// File/Function Blocks/FB_FileHandlerBase
FUNCTION_BLOCK ABSTRACT FB_FileHandlerBase EXTENDS FB_Component<GC_File.INDEX_COMMAND_MIN,GC_File.INDEX_COMMAND_MAX > IMPLEMENTS I_FileHandlerBaseConfiguration
VAR
    FileHandlerConfiguration		: ST_FileHandlerConfiguration;
    FileHandlerStatus      			: ST_FileHandlerBaseStatus;
END_VAR

PROPERTY P_FileHandlerBaseConfiguration : REFERENCE TO ST_FileHandlerConfiguration
GET
P_FileHandlerBaseConfiguration REF= FileHandlerConfiguration;
END_GET
END_PROPERTY

METHOD PROTECTED _InitializeReferences : BOOL
//Initialize data references
//Order is important!
BaseConfiguration.InstancePath 						REF= InstancePath;

ComponentConfiguration.BaseConfiguration 			REF= SUPER^.BaseConfiguration;
                                                    
ComponentStatus.BaseStatus							REF= SUPER^.BaseStatus;
                                                    
//SUPER^.ComponentStatus.LastCommandStatus			REF= SUPER^.Commands[GC_File.INDEX_COMMAND_MIN].P_CommandStatus;

ComponentStatus.AmsNetId							REF= ComponentConfiguration.AmsNetId;

FileHandlerConfiguration.ComponentConfiguration		REF= SUPER^.ComponentConfiguration;

FileHandlerStatus.ComponentStatus					REF= SUPER^.ComponentStatus;

_InitializeReferences 								:= TRUE; // apply at end of all reference initialization
END_METHOD

METHOD CyclicLogic
SUPER^.CyclicLogic();
END_METHOD

{warning 'Add property implementation'}
PROPERTY P_FileHandlerBaseStatus : REFERENCE TO ST_FileHandlerBaseStatus
GET
P_FileHandlerBaseStatus REF= FileHandlerStatus;
END_GET
END_PROPERTY

END_FUNCTION_BLOCK

// File/Interfaces/I_FileHandlerBaseConfiguration
INTERFACE I_FileHandlerBaseConfiguration EXTENDS __SYSTEM.IQueryInterface

PROPERTY P_FileHandlerBaseConfiguration : REFERENCE TO ST_FileHandlerConfiguration
GET
END_GET
END_PROPERTY

END_INTERFACE

// File/Function Blocks/FB_FileHandlerJson
{attribute 'no_explicit_call' := 'do not call this POU directly'}
FUNCTION_BLOCK FB_FileHandlerJson EXTENDS FB_FileHandlerBase IMPLEMENTS I_FileHandlerJson
VAR
	JsonReadWriteDatatype			: Tc3_JsonXml.FB_JsonReadWriteDatatype;
	JsonDomParser					: Tc3_JsonXml.FB_JsonDomParser;
	JsonSaxWriter					: Tc3_JsonXml.FB_JsonSaxWriter;
END_VAR

{error 'Add method implementation or delete method to use base implementation'}
METHOD CyclicLogic
END_METHOD

END_FUNCTION_BLOCK

// File/Interfaces/I_FileHandlerJson
INTERFACE I_FileHandlerJson EXTENDS I_FileHandlerBase

END_INTERFACE

// File/Interfaces/I_FileHandlerBase
INTERFACE I_FileHandlerBase EXTENDS I_BaseCyclic

METHOD AppendToFileByPointer : I_FileHandlerBase
VAR_INPUT
	pContent 	: PVOID; //Pointer to Content
//	nContent	: UDINT; //Size of Content
	nElement	: INT; //Size of Content Element
END_VAR
END_METHOD

METHOD CloseFile : I_FileHandlerBase
END_METHOD

METHOD CreateFile : I_FileHandlerBase
VAR_INPUT
	Mode	: DWORD := Tc2_System.Global_Variables.FOPEN_MODEAPPEND; //i.e., Tc2_System.Global_Variables.FOPEN_MODEAPPEND, otherwise 0!
END_VAR
END_METHOD

METHOD DeleteFile : I_FileHandlerBase
END_METHOD

METHOD OpenFile : I_FileHandlerBase
END_METHOD

METHOD ReadFromFile : I_FileHandlerBase
END_METHOD

METHOD RenameFile : I_FileHandlerBase
VAR_INPUT
	OldName : T_MaxString;
	NewName : T_MaxString;	
END_VAR
END_METHOD

METHOD WriteFile : I_FileHandlerBase
END_METHOD

PROPERTY P_FileHandlerBaseStatus : REFERENCE TO ST_FileHandlerBaseStatus
GET
END_GET
END_PROPERTY

END_INTERFACE

// File/Interfaces/I_FileHandlerCsv
INTERFACE I_FileHandlerCsv EXTENDS I_FileHandlerBase

METHOD AppendToFileByString : I_FileHandlerCsv
VAR_INPUT
	sContent 	: Tc2_System.T_MaxString;
END_VAR
END_METHOD

METHOD AppendToFileBySystimeString : I_FileHandlerCsv
VAR_INPUT
	sContent 	: ST_SystimeString;
END_VAR
END_METHOD

PROPERTY P_AppendRingBufferStatus : REFERENCE TO ST_RingBufferStatus
GET
END_GET
END_PROPERTY

PROPERTY P_FileHandlerCsvStatus : REFERENCE TO ST_FileHandlerCSVStatus
GET
END_GET
END_PROPERTY

END_INTERFACE

// Functions/Numbers/F_MapLREAL
FUNCTION F_MapLREAL : LREAL
VAR_INPUT
    x       : LREAL;
    in_min  : LREAL;
    in_max  : LREAL;
    out_min : LREAL;
    out_max : LREAL;
END_VAR

IF (in_max - in_min) <> 0 THEN
	F_MapLReal := (((x - in_min) * (out_max - out_min)) / (in_max - in_min)) + out_min;
ELSE
	// fallback if input range is zero
	F_MapLREAL := out_min;
END_IF;

END_FUNCTION

// Functions/Strings/F_GetAllButFirstWord
FUNCTION F_GetAllButFirstWord : Tc2_System.T_MaxString
VAR_INPUT
    sInput : Tc2_System.T_MaxString;
END_VAR
VAR
    i           : INT;
    strLength   : INT;
    bChar       : BYTE := 32; // ASCII for space ' '
    arrInput    : ARRAY[0..255] OF BYTE;
    startCopy   : INT := -1;
    resultStr   : Tc2_System.T_MaxString := '';
END_VAR

strLength := LEN(sInput);
arrInput := Tc2_Utilities.MAXSTRING_TO_BYTEARR(sInput); // Convert to BYTE array

// Find first space
FOR i := 0 TO strLength - 1 DO
    IF arrInput[i] = bChar THEN
        startCopy := i + 1; // index after the space
        EXIT;
    END_IF
END_FOR

// If no space found or nothing after space, return empty
IF (startCopy = -1) OR (startCopy >= strLength) THEN
    F_GetAllButFirstWord := '';
    RETURN;
END_IF

// Skip additional spaces (if any)
WHILE (startCopy < strLength) AND (arrInput[startCopy] = bChar) DO
    startCopy := startCopy + 1;
END_WHILE

// Build result from the rest of the string
FOR i := startCopy TO strLength - 1 DO
    resultStr := Tc2_Standard.CONCAT(resultStr, Tc2_System.F_ToCHR(arrInput[i]));
END_FOR

F_GetAllButFirstWord := resultStr;

END_FUNCTION

// Functions/Strings/F_GetFirstWordInString
FUNCTION F_GetFirstWordInString : Tc2_System.T_MaxString
VAR_INPUT
    sInput : Tc2_System.T_MaxString; // Input string like '0 NA' or '-15000 NA'
	TerminationChar	: BYTE := 32; // ASCII for space ' '
END_VAR
VAR
    i           : INT;
    strLength   : INT;
    resultStr   : Tc2_System.T_MaxString;
    arrInput    : ARRAY[0..255] OF BYTE;
END_VAR

strLength := LEN(sInput);
arrInput := Tc2_Utilities.MAXSTRING_TO_BYTEARR(sInput); // Convert to BYTE array

// If first char is space or string is empty, return empty
IF (strLength = 0) OR (arrInput[0] = TerminationChar) THEN
    F_GetFirstWordInString := '';
    RETURN;
END_IF

// Build result from left until first space
resultStr := '';
FOR i := 0 TO strLength DO
    IF arrInput[i] = TerminationChar THEN
        EXIT;
    END_IF
    resultStr := Tc2_Standard.CONCAT(resultStr, Tc2_System.F_ToCHR(arrInput[i]));
END_FOR

F_GetFirstWordInString := resultStr;

END_FUNCTION

// Functions/Strings/F_ReplaceInString
FUNCTION F_ReplaceInString : STRING
VAR_INPUT
  ObjectString    : STRING;
  StringToRemove  : STRING;
  StringToInsert  : STRING;
END_VAR
VAR
  tempString      : STRING;
  ReplacePosn     : INT;
END_VAR

tempString  := ObjectString;

WHILE(Tc2_Standard.FIND(STR1 := tempString, STR2 := StringToRemove) <> 0) DO
  ReplacePosn := Tc2_Standard.FIND(STR1 := tempString, STR2 := StringToRemove);
  tempString  := Tc2_Standard.REPLACE(L := Tc2_Standard.LEN(STR := StringToRemove), P := ReplacePosn,
                                      STR1 := tempString, STR2 := StringToInsert);
END_WHILE

F_ReplaceInString   := tempString;

END_FUNCTION

// Functions/Strings/F_TrimString
FUNCTION F_TrimString : Tc2_System.T_MaxString
VAR_INPUT
	InputString		: Tc2_System.T_MaxString;
	Prefix			: Tc2_System.T_MaxString := '$R';
	Suffix			: Tc2_System.T_MaxString := '$N';
END_VAR
VAR
	FindCRPosnInString	: INT;
END_VAR

// Capture string to trim
F_TrimString := InputString;

// Remove prefix - if found
FindCRPosnInString := Tc2_Standard.FIND(STR1 := F_TrimString, STR2 := Prefix);
IF FindCRPosnInString <> 0 THEN
	F_TrimString := Tc2_Standard.DELETE(STR := F_TrimString, LEN := Tc2_Standard.LEN(Prefix), POS := FindCRPosnInString);
END_IF

// Remove suffix - if found
FindCRPosnInString := Tc2_Standard.FIND(STR1 := F_TrimString, STR2 := Suffix);
IF FindCRPosnInString <> 0 THEN
	F_TrimString := Tc2_Standard.DELETE(STR := F_TrimString, LEN := Tc2_Standard.LEN(Suffix), POS := FindCRPosnInString);
END_IF

END_FUNCTION

// Functions/Time/F_DateTimeConvertedAsT_MaxString
FUNCTION F_DateTimeConvertedAsT_MaxString : Tc2_System.T_MaxString
VAR_INPUT
  HourDeltaUTC              : SINT  := GPL_Base.HourDeltaFromUtc;
END_VAR
VAR
  timeAsFileTime            : Tc2_Utilities.T_FILETIME64;
  tempDtForUtcCalc          : Tc2_Utilities.T_FILETIME64;
END_VAR
VAR CONSTANT
  CountOf100NsIncrement1Hr  : LINT  := 36000000000;
END_VAR

timeAsFileTime    := Tc2_System.F_GetSystemTime();

tempDtForUtcCalc  := timeAsFileTime + (HourDeltaUTC * GC.CountOf100NsIncrement1Hr);

F_DateTimeConvertedAsT_MaxString := F_FileTimeToString(tempDtForUtcCalc);

END_FUNCTION

// Functions/Time/F_SystemTimeUtcCorrected
FUNCTION F_SystemTimeUtcCorrected : ULINT
VAR_INPUT
  HourDeltaUTC              : SINT  := GPL_Base.HourDeltaFromUtc;
END_VAR
VAR
  timeAsFileTime            : Tc2_Utilities.T_FILETIME64;
  tempDtForUtcCalc          : Tc2_Utilities.T_FILETIME64;
END_VAR

timeAsFileTime            := Tc2_System.F_GetSystemTime();
                          
tempDtForUtcCalc          := timeAsFileTime + (HourDeltaUTC * GC_Base.CountOf100NsIncrement1Hr);

F_SystemTimeUtcCorrected    := tempDtForUtcCalc;

END_FUNCTION

// Hashing/ITFs/I_HashTableExt
INTERFACE I_HashTableExt EXTENDS I_HashTableBase

//— True if name is present (fast path)
METHOD PUBLIC Contains : BOOL
VAR_INPUT
  NameIn : T_MaxString;
END_VAR
END_METHOD

METHOD OnLoadFactorExceeded
VAR
  Message : T_MaxString;
END_VAR
END_METHOD

//— Double the table size and re‐insert all live entries
METHOD PUBLIC Rehash : VOID
VAR
  oldKeys    : ARRAY[0..1023] OF T_MaxString;
  oldVals    : ARRAY[0..1023] OF UDINT;
  oldCap     : UINT;
  i : UINT;
END_VAR
END_METHOD

//— Remove an entry (marks a tombstone)
METHOD PUBLIC Remove : BOOL
VAR_INPUT
  NameIn : T_MaxString;
END_VAR
VAR
  slot, start : UINT;
END_VAR
END_METHOD

END_INTERFACE

// PRGs/PRG_LOG
PROGRAM PRG_LOG

// Simple call - if GVL_System doesn't exist in the project, PRG_LOG shouldn't be included either
// Both should be part of the base library package
GVL_System.EventLogHandler.CyclicLogic();

END_PROGRAM

// PRGs/PRG_PRETEST
PROGRAM PRG_PRETEST
VAR
//	Sequencer							: FB_PackMLSequencer;
	
	TrigStart			: BOOL;
	TrigStop			: BOOL;
	TrigAbort			: BOOL;

	InitComplete						: BOOL;
	
//File Testing
// 	FileHandlerCsv						: FB_FileHandlerCsvConfigured;
// 	iFileHandlerCsv						: I_FileHandlerCsv := FileHandlerCsv;
	
	CommandUnderTest					: FB_CommandUnderTest;
	CommandConfiguration				: FB_CmdPermIntlkConfiguration;
	iCommandConfiguration				: I_CommandConfiguration := CommandConfiguration;
	CommandStatus						: ST_CommandStatus;
	
	Debounce							: FB_Debounce;
	iDebounce							: I_Debounce := Debounce;
	iDebounceCfg						: I_DebounceConfiguration := Debounce;
	TrigDebounceCfg						: BOOL;
	TrigDebounceT						: BOOL;
	TrigDebounceF						: BOOL;
	
	TrigCreateFile			: BOOL;
	TrigRenameFile			: BOOL;
	TrigDeleteFile			: BOOL;
	TrigAppendToFile		: BOOL;
	TrigCloseFile			: BOOL;
	TrigReadFromFile		: BOOL;
	TrigWriteFile			: BOOL;
	TrigOpenFile			: BOOL;
	
	TrigCmdConfig			: BOOL;
	TrigCmdStatus			: BOOL;
END_VAR

//IF GVL_System.PlcSystemInfo[GPL_Base.INDEX_LOG_TASK].FirstCycle THEN
IF NOT __ISVALIDREF(GVL_System.EventLogHandler.EventLogHandlerConfiguration.BaseConfiguration) THEN
	GVL_System.EventLogHandler.Initialize();
	RETURN;
END_IF

Debounce.CyclicLogic();

IF iDebounceCfg <> 0 THEN
	IF TrigDebounceCfg THEN
		iDebounceCfg.P_DebounceConfiguration.tOnDelay	:= T#3S;
		iDebounceCfg.P_DebounceConfiguration.tOffDelay	:= T#3S;
		iDebounceCfg.P_DebounceConfiguration.BaseConfiguration.InSimulation	:= true;
		TrigDebounceCfg	:= FALSE;
	END_IF
END_IF

IF iDebounce <> 0 THEN
	IF TrigDebounceT THEN
		iDebounce.P_RawSignal	:= TRUE;
		TrigDebounceT	:= FALSE;
	END_IF
	IF TrigDebounceF THEN
		iDebounce.P_RawSignal	:= FALSE;
		TrigDebounceF	:= FALSE;
	END_IF
END_IF

// Sequencer.CyclicLogic();
// 
// IF TrigStart THEN
// 	Sequencer.Start();
// 	TrigStart	:= FALSE;
// END_IF
// 
// IF TrigStop THEN
// 	Sequencer.Stop();
// 	TrigStop	:= FALSE;
// END_IF
// 
// IF TrigAbort THEN
// 	Sequencer.Abort();
// 	TrigAbort	:= FALSE;
// END_IF

IF TrigCmdConfig THEN
	iCommandConfiguration.P_CommandConfiguration.CommandDescription := 'yonkers';
	iCommandConfiguration.P_CommandConfiguration.Priority := E_CommandPriority.Priority_High;
	iCommandConfiguration.P_CommandConfiguration.RetryCountONLYFORCOMMSENDS	:= 12;
	CommandUnderTest.SetCommandConfiguration(ConfigurationToSet := iCommandConfiguration);
	TrigCmdConfig := FALSE;
END_IF

IF TrigCmdStatus THEN
	CommandStatus.CommandTryCount := 11;
	CommandStatus.StepState := E_CommandState.Paused;
	CommandUnderTest.SetCommandStatus(DesiredBaseStatus := CommandStatus);
	TrigCmdStatus := FALSE;
END_IF

// IF iFileHandlerCsv <> 0 THEN
// 	iFileHandlerCsv.CyclicLogic();
// END_IF
// 
// IF iFileHandlerCsv <> 0 THEN
// 	
// 	IF TrigCreateFile THEN
// 		iFileHandlerCsv.CreateFile();
// 		TrigCreateFile := FALSE;
// 	END_IF
// 	
// 	IF TrigRenameFile THEN
// 		iFileHandlerCsv.RenameFile(OldName := 'Log_133978534968790000x.csv', NewName := 'abc_133978534968790000x.csv');
// 		TrigRenameFile := FALSE;
// 	END_IF
// 	
// 	IF TrigDeleteFile THEN
// 		iFileHandlerCsv.DeleteFile();
// 		TrigDeleteFile := FALSE;
// 	END_IF
// 	
// 	IF TrigAppendToFile THEN
// 		//iFileHandlerCsv.AppendToFileByPointer(pContent := , nElement := );
// 		TrigAppendToFile := FALSE;
// 	END_IF
// 	
// 	IF TrigCloseFile THEN
// 		iFileHandlerCsv.CloseFile();
// 		TrigCloseFile := FALSE;
// 	END_IF
// 	
// 	IF TrigReadFromFile THEN
// 		//iFileHandlerCsv.ReadFromFile();
// 		TrigReadFromFile := FALSE;
// 	END_IF
// 	
// 	IF TrigWriteFile THEN
// 		//iFileHandlerCsv.WriteFile();
// 		TrigWriteFile := FALSE;
// 	END_IF
// 	
// 	IF TrigOpenFile THEN
// 		iFileHandlerCsv.OpenFile();
// 		TrigOpenFile := FALSE;
// 	END_IF
// 	
// END_IF

END_PROGRAM

// Tests/MockFBs/FB_CommandUnderTest
{attribute 'no_explicit_call' := 'do not call this POU directly'}
FUNCTION_BLOCK FB_CommandUnderTest EXTENDS FB_Command IMPLEMENTS I_CommandUnderTest

METHOD SetCommandConfiguration
VAR_INPUT
	ConfigurationToSet	: REFERENCE TO I_CommandConfiguration;
END_VAR
SUPER^._iCommandConfiguration := ConfigurationToSet;
END_METHOD

METHOD SetCommandStatus
VAR_INPUT
	DesiredBaseStatus	: REFERENCE TO ST_CommandStatus;
END_VAR
SUPER^.CommandStatus := DesiredBaseStatus;
END_METHOD

END_FUNCTION_BLOCK

// Tests/TestInterfaces/I_CommandUnderTest
INTERFACE I_CommandUnderTest EXTENDS I_Command

METHOD SetCommandStatus
VAR_INPUT
	DesiredBaseStatus				: REFERENCE TO ST_CommandStatus;
END_VAR
END_METHOD

END_INTERFACE

// PRGs/PRG_TEST
PROGRAM PRG_TEST
VAR
//	RingBufferTests							: FB_RingBufferTests; //OK
	
//	StringTests								: FB_StringParsingFunctionTests; //OK
	
//	HashTableTests							: FB_HashTableTests; //OK

//	BaseStaticTests							: FB_BaseStaticTests; //OK
	
//	BaseCyclicTests							: FB_BaseCyclicTests; //OK
	
//	DebounceTests							: FB_DebounceTests; //OK

//	PermIntlkTests							: FB_PermIntlkTests; //OK
	
//	CommandTests							: FB_CommandTestsI; //can cause stack overflow running more than one of these FBs at a time;
	
//	CommandTestsII							: FB_CommandTestsII; //can cause stack overflow - likely a result of logger issue, but untested
	
//	CommandTestsIII							: FB_CommandTestsIII; //can cause stack overflow - likely a result of logger issue, but untested
	
//	CommandTestsIV							: FB_CommandTestsIV; //can cause stack overflow - likely a result of logger issue, but untested

//	CommandTestsV							: FB_CommandTestsV; //can cause stack overflow - likely a result of logger issue, but untested
	
//	CommandTestsVI							: FB_CommandTestsVI; //can cause stack overflow - likely a result of logger issue, but untested

	CommandTestsVII							: FB_CommandTestsVII;
	
//	ComponentTests							: FB_ComponentTests; //OK
	
//	SequencerTests							: FB_SequencerTests; //OK
	
//	LogTests								: FB_LogTests; //suspect stack overflow?

//	RingBufferLoggerTests					: FB_RingBufferLoggerTests; //untested
END_VAR

//IF GVL_System.PlcSystemInfo[GPL_Base.INDEX_LOG_TASK].FirstCycle THEN
IF NOT __ISVALIDREF(GVL_System.EventLogHandler.EventLogHandlerConfiguration.BaseConfiguration) THEN
	GVL_System.EventLogHandler.Initialize();
	RETURN;
END_IF

TcUnit.RUN();

END_PROGRAM

// Tests/FB_RingBufferTests
FUNCTION_BLOCK FB_RingBufferTests EXTENDS TcUnit.FB_TestSuite
VAR
    i : DINT; //FOR loop index
    PointerBefore : PVOID;
    PointerAfter : PVOID;
    // Array instances for test methods (indices 0-57)
    RingBuffer : ARRAY[GC_Test.INDEX_TestFB_RingBuffer_MIN..GC_Test.INDEX_TestFB_RingBuffer_MAX] OF FB_RingBufferKeyString;
END_VAR

GivenAdd3ObjectExpect3ObjectToBeAdded();
GivenAdd3Remove3ExpectFifoOrder();
GivenAddAndRemoveAlternateExpectFIFOOrder();
GivenAddExactCapacityThenRemoveAllExpectFIFO();
GivenAddMoreThanDoubleCapacityThenReadAllExpectOnlyRecent();
GivenRapidAddRemoveInLoopExpectCorrectFinalCount();
GivenAddObjectExpectStatusFlagsUpdateCorrectly();
GivenAddObjectLength10ExpectObjectToBeAdded();
GivenAddObjectLength20ExpectObjectToBeAdded();
GivenAddObjectLength40ExpectObjectToBeAdded();
GivenAddObjectLength80ExpectObjectToBeAdded();
GivenAddRemoveOneObjectExpectSameObjectBack();
GivenAddThenClearLastRemovedExpectEmptyFlag();
GivenAddThenQueryPointerConsistency();
GivenAddThenReadExpectSameObject();
GivenAddWhileRemoveInProgressExpectNoCorruption();
GivenAddWithinvalidRefExpectNoWrite();
GivenClearBufferExpectObjectCountZero();
GivenClearCalledExpectallStatsReset();
GivenEmptyBufferExpectPeekReturnsDefault();
GivenFullBufferAddOneExpectOverwriteOldest();
GivenLargeStringExpectTruncationOrError();
GivenMultipleAddinSingleCycleExpectAllStored();
GivenMultipleAddsSameCycleExpectAllStored();
GivenMultipleObjectsExpectPeekAlwaysReturnsFirst();
GivenNullRefInputExpectGracefulHandling();
GivenOneObjectAddedExpectPeekReturnsit();
GivenOversizedObjectExpectPartialWriteOrError();
GivenOverwriteOccursExpectOnlyRecentN();
GivenOverwriteThenReadExpectMostRecent();
GivenPeekThenClearPeekedFlagExpectReset();
GivenReadFromEmptyExpectNoCrashOrInvalid();
GivenReadThenClearStatusExpectFlagsReset();
GivenRemoveFromEmptyExpectError();
GivenRemoveObjectExpectLastRemovedMatchesExpected();
GivenRemoveOnEmptyExpectNoCrash();
GivenRemovePointerWrapsAroundExpectValidRead();
GivenRemoveThenReadExpectNoNewData();
GivenUpdateRemovePointerBoundaryExpectCorrectWrap();
GivenUpdateWritePointerBoundaryExpectCorrectWrap();
GivenWrapAroundReadPointerExpectCorrectRead();
GivenWrapAroundWriteExpectValidRead();
GivenWritePointerWrapsAroundExpectValidOverwrite();
GivenZeroCapacityBufferExpectNoWrite();
GivenInitExpectDefaultPointerAndState();
GivenAddThenRemoveExpectCorrectCounters();
GivenFillBufferExpectIsFullTrue();
GivenAddRemoveExpectFlagsSet();
GivenPeekAndReadExpectFlagsSet();
GivenOverwriteExpectFlagSet();
GivenAddExpectCorrectByteCount();
Test_BufferStatus_AfterAddAndRemove();
Test_BufferStatus_Add4Remove2();
GivenOverwriteThenRemoveExpectOverwriteCleared();
GivenAddMoreThanCapacityExpectCorrectGlobalCounter();
GivenReadThenRemoveExpectCorrectFlagsAndCounts();

METHOD PRIVATE GivenAdd3ObjectExpect3ObjectToBeAdded
VAR
    TestObject      : ST_SystimeString := (stringval := 'HelloWorld');  
END_VAR
TEST(__POUNAME());

RingBuffer[0].Initialize();
RingBuffer[0].AddObject(RefObject := TestObject);
RingBuffer[0].AddObject(RefObject := TestObject);
RingBuffer[0].AddObject(RefObject := TestObject);

AssertEquals_UDINT(Actual := RingBuffer[0].RingBufferStatus.GlobalCounter, Expected := 3, 
            Message := 'Expected matching counts');

TEST_FINISHED();
END_METHOD

METHOD PRIVATE GivenAdd3Remove3ExpectFifoOrder
VAR
  Obj1 : ST_SystimeString := (stringval := 'One');
  Obj2 : ST_SystimeString := (stringval := 'Two');
  Obj3 : ST_SystimeString := (stringval := 'Three');
  Removed : ST_SystimeString;
END_VAR
TEST(__POUNAME());

RingBuffer[1].Initialize();
RingBuffer[1].AddObject(RefObject := Obj1);
RingBuffer[1].AddObject(RefObject := Obj2);
RingBuffer[1].AddObject(RefObject := Obj3);

RingBuffer[1].RemoveObject(); Removed := RingBuffer[1].LastObjRemoved;
AssertEquals(Actual := Removed.stringval, Expected := Obj1.stringval, Message := 'First item should be "One"');

RingBuffer[1].RemoveObject(); Removed := RingBuffer[1].LastObjRemoved;
AssertEquals(Actual := Removed.stringval, Expected := Obj2.stringval, Message := 'Second item should be "Two"');

RingBuffer[1].RemoveObject(); Removed := RingBuffer[1].LastObjRemoved;
AssertEquals(Actual := Removed.stringval, Expected := Obj3.stringval, Message := 'Third item should be "Three"');

TEST_FINISHED();
END_METHOD

METHOD PRIVATE GivenAddAndRemoveAlternateExpectFIFOOrder
VAR
    TestObject : ST_SystimeString := (stringval := 'Hello');
    Removed    : ST_SystimeString;
END_VAR
TEST(__POUNAME());

RingBuffer[2].Initialize();
RingBuffer[2].AddObject(RefObject := TestObject);
RingBuffer[2].RemoveObject(); Removed := RingBuffer[2].LastObjRemoved;
AssertEquals(Actual := Removed.stringval, Expected := TestObject.stringval,
    Message := 'Expected same object after alternate add/remove');
TEST_FINISHED();
END_METHOD

METHOD PRIVATE GivenAddExactCapacityThenRemoveAllExpectFIFO
VAR
    Capacity   : UDINT := RingBuffer[3].RingBufferStatus.BufferCapacity;
    i          : UDINT;
    Expected   : ST_SystimeString;
    Removed    : ST_SystimeString;
END_VAR
TEST(__POUNAME());

RingBuffer[3].Initialize();
Capacity := RingBuffer[3].RingBufferStatus.BufferCapacity;

// Add Capacity number of unique objects
FOR i := 1 TO Capacity DO
    Expected.stringval := CONCAT('Item', UDINT_TO_STRING(i));
    RingBuffer[3].AddObject(RefObject := Expected);
END_FOR

// Remove and verify FIFO order
FOR i := 1 TO Capacity DO
    RingBuffer[3].RemoveObject();
    Removed := RingBuffer[3].LastObjRemoved;
    Expected.stringval := CONCAT('Item', UDINT_TO_STRING(i));
    AssertEquals(Actual := Removed.stringval, Expected := Expected.stringval,
        Message := CONCAT('Expected FIFO order, mismatch at item ', UDINT_TO_STRING(i)));
END_FOR

TEST_FINISHED();
END_METHOD

METHOD PRIVATE GivenAddExpectCorrectByteCount
VAR
    TestObject  : ST_SystimeString := (stringval := 'ByteCountTest');
    Expected    : ULINT;
END_VAR
TEST(__POUNAME());

RingBuffer[4].Initialize();
RingBuffer[4].AddObject(RefObject := TestObject);
Expected := RingBuffer[4].RingBufferConfiguration.ByteCountOfDataObj;

AssertEquals(
    Actual := RingBuffer[4].RingBufferStatus.ByteCountInBufferPrim,
    Expected := Expected,
    Message := 'Expected ByteCountInBufferPrim = ByteCountOfDataObj * 1'
);

TEST_FINISHED();
END_METHOD

METHOD PRIVATE GivenAddMaxUDINTObjectsExpectGracefulHandling
VAR
    TestObject : ST_SystimeString := (stringval := 'Hello');
    Removed    : ST_SystimeString;
END_VAR
TEST(__POUNAME());

FOR i := 1 TO 100 DO
    RingBuffer[5].AddObject(RefObject := TestObject);
END_FOR

AssertTrue(Condition := RingBuffer[5].RingBufferStatus.GlobalCounter <= 100, Message := 'Buffer overflowed UDINT max unexpectedly');

TEST_FINISHED();
END_METHOD

METHOD PRIVATE GivenAddMoreThanCapacityExpectCorrectGlobalCounter
VAR
	DummyObj     : ST_SystimeString;
	i            : INT;
	capacity     : UDINT;
	testval80	: UDINT := 80;
END_VAR
TEST(__POUNAME());

RingBuffer[6].Initialize();
RingBuffer[6].ClearBuffer();
capacity := RingBuffer[6].RingBufferStatus.BufferCapacity;

// Add more than capacity
FOR i := 1 TO 10 DO
	RingBuffer[6].AddObject(RefObject := DummyObj);
END_FOR

AssertEquals(capacity, RingBuffer[6].RingBufferStatus.GlobalCounter, 'Expected GlobalCounter to cap at capacity');
//AssertEquals(Expected := (testval80 * capacity), RingBuffer[6].RingBufferStat.ByteCountInBufferPrim, 'Expected ByteCount = capacity * size');
AssertTrue(RingBuffer[6].RingBufferStatus.Overwriting, 'Expected Overwriting = TRUE');

TEST_FINISHED();
END_METHOD

METHOD PRIVATE GivenAddMoreThanDoubleCapacityThenReadAllExpectOnlyRecent
VAR
    Capacity     : UDINT := RingBuffer[7].RingBufferStatus.BufferCapacity;
    TotalAdds    : UDINT := Capacity * 2 + 1;
    i            : UDINT;
    TestObject   : ST_SystimeString;
    Removed      : ST_SystimeString;
    ExpectedIdx  : UDINT;
    Expected     : ST_SystimeString;
END_VAR
TEST(__POUNAME());

// Add more than double the capacity worth of uniquely identifiable objects
FOR i := 1 TO TotalAdds DO
    TestObject.stringval := CONCAT('Item', UDINT_TO_STRING(i));
    RingBuffer[7].AddObject(RefObject := TestObject);
END_FOR

// Only the most recent [Capacity] elements should be stored, starting from TotalAdds - Capacity + 1
FOR i := 1 TO Capacity DO
    RingBuffer[7].RemoveObject();
    Removed := RingBuffer[7].LastObjRemoved;
    ExpectedIdx := TotalAdds - Capacity + i;
    Expected.stringval := CONCAT('Item', UDINT_TO_STRING(ExpectedIdx));
    AssertEquals(Actual := Removed.stringval, Expected := Expected.stringval,
        Message := CONCAT('Expected retained item: ', Expected.stringval));
END_FOR

TEST_FINISHED();
END_METHOD

METHOD PRIVATE GivenAddObjectExpectStatusFlagsUpdateCorrectly
VAR
    TestObject : ST_SystimeString := (stringval := 'StatusCheck');
END_VAR
TEST(__POUNAME());

RingBuffer[8].Initialize();

